# B&R Automation Studio project DuctLines (part 11)

#### Cyclic.ld
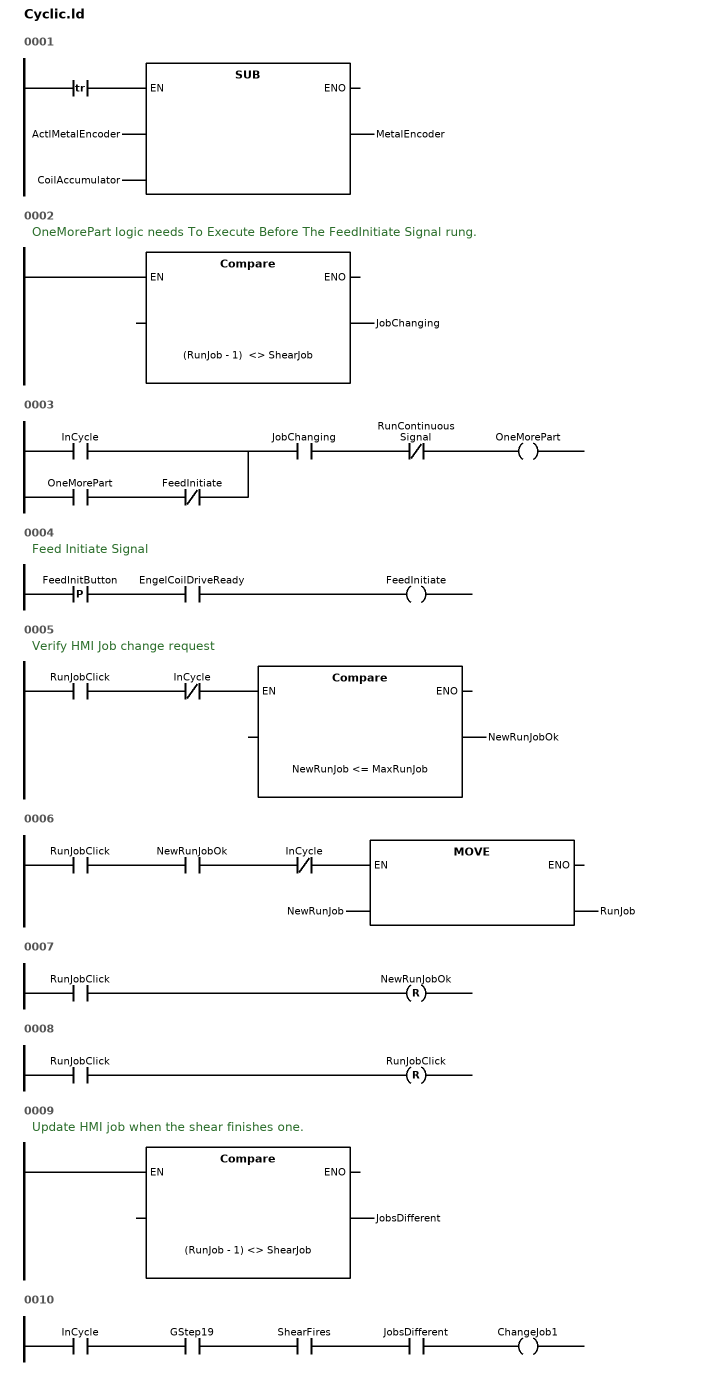
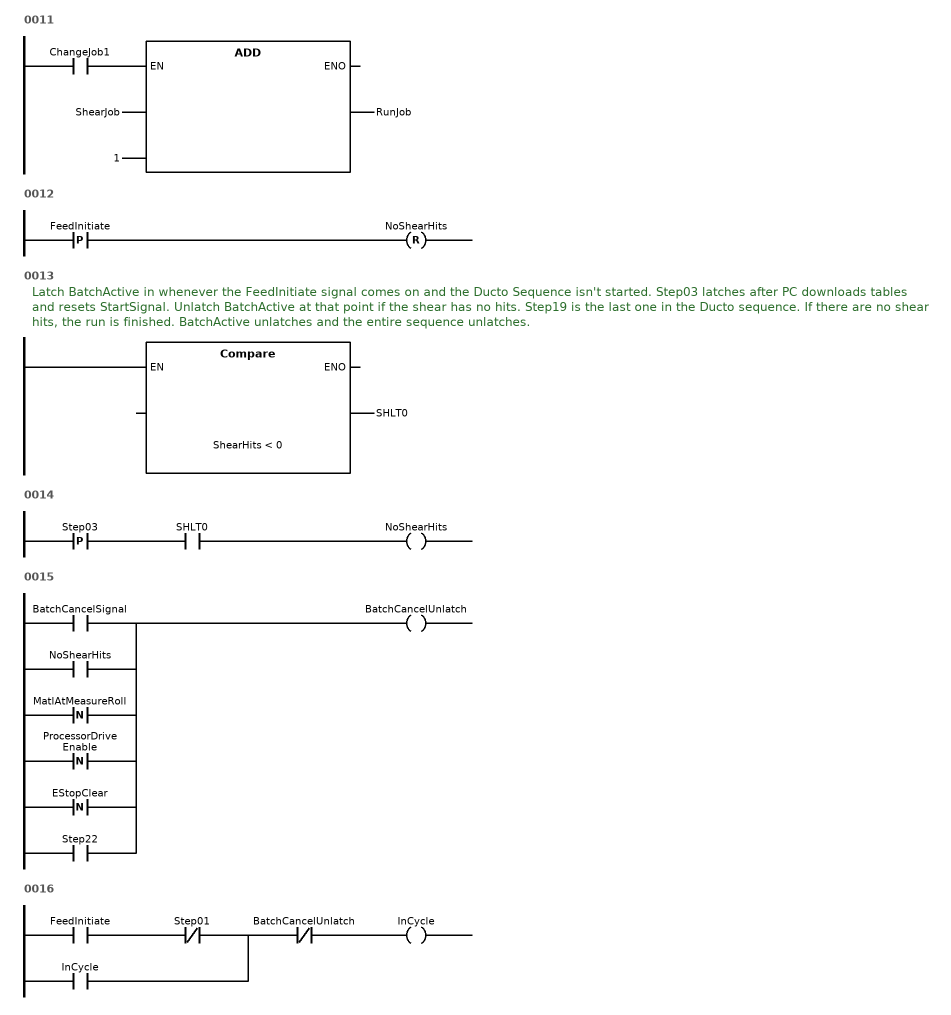
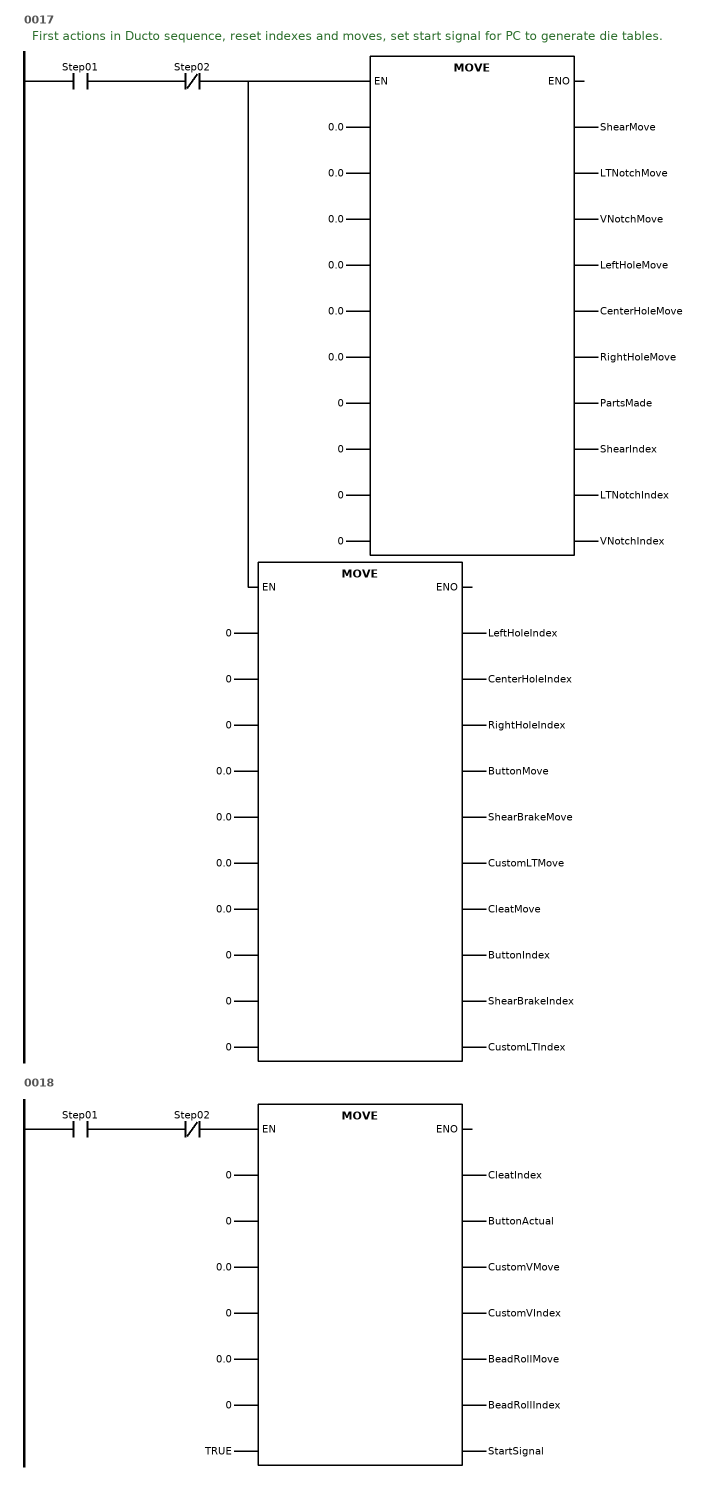
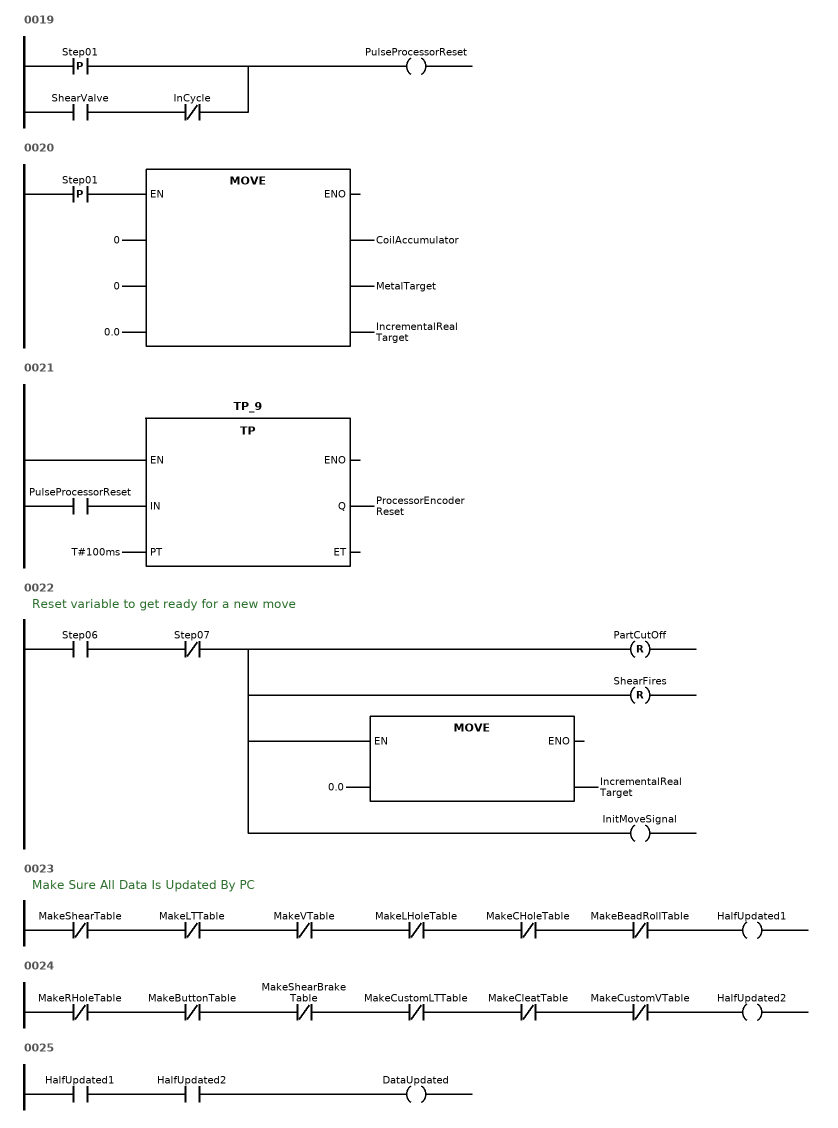
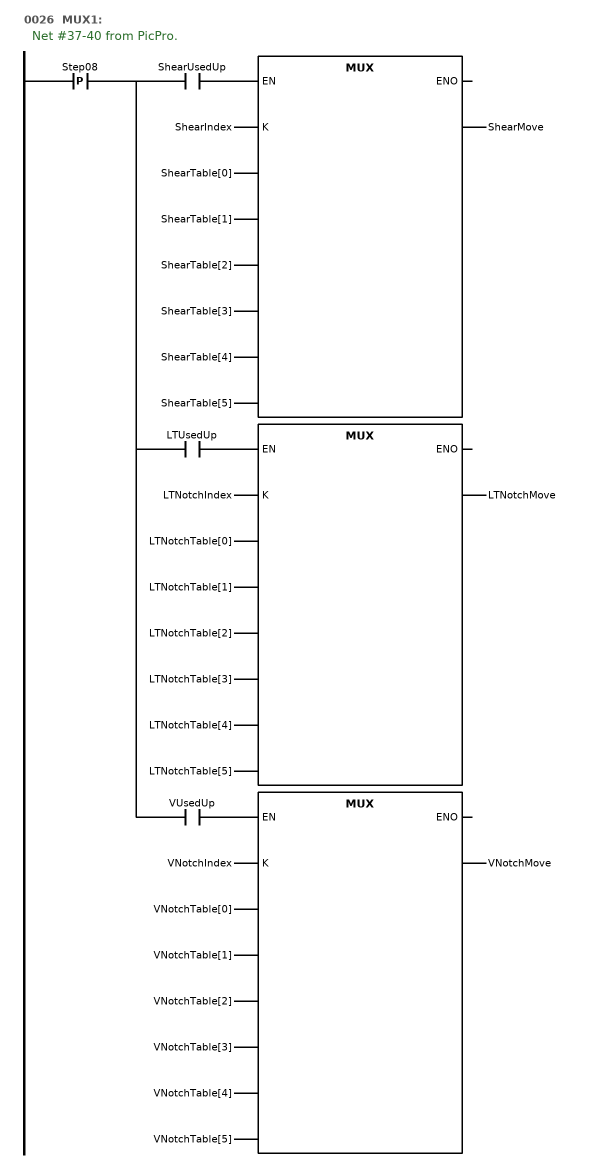
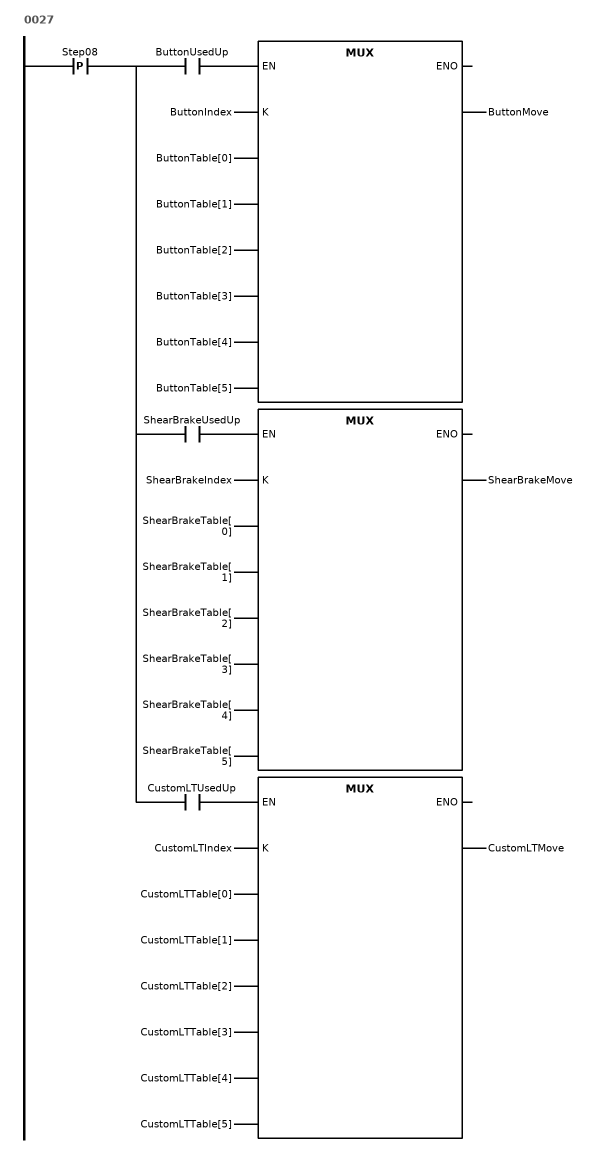
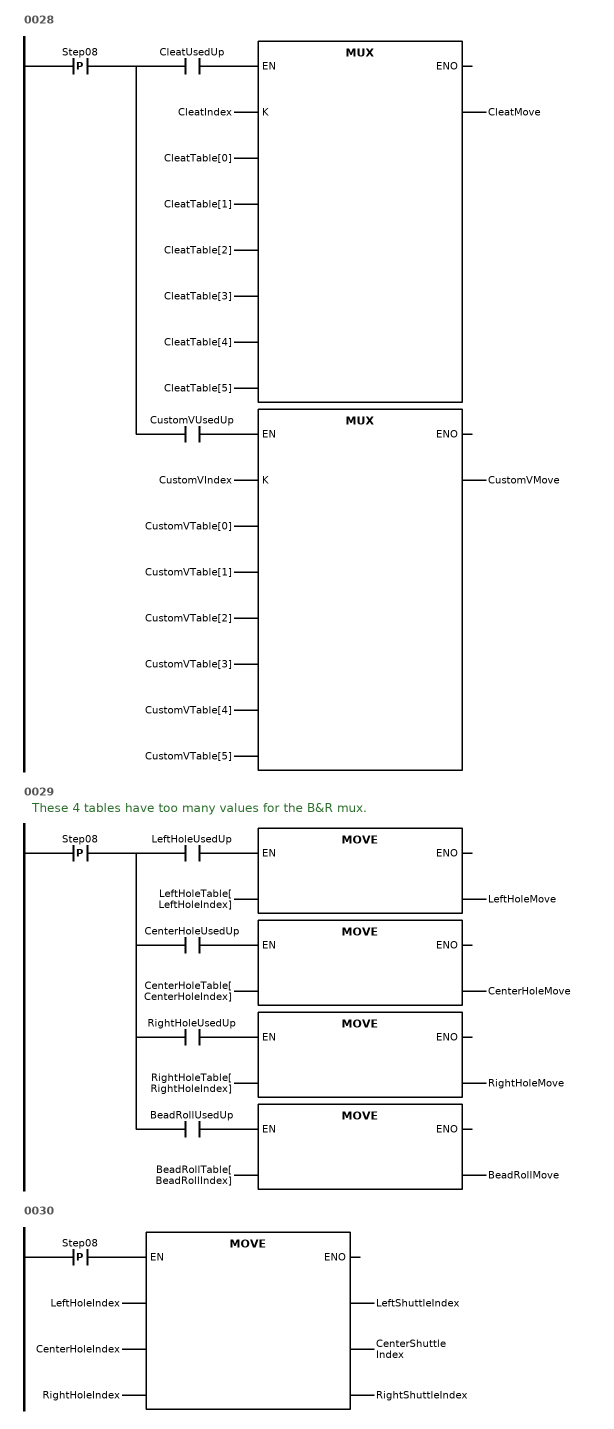
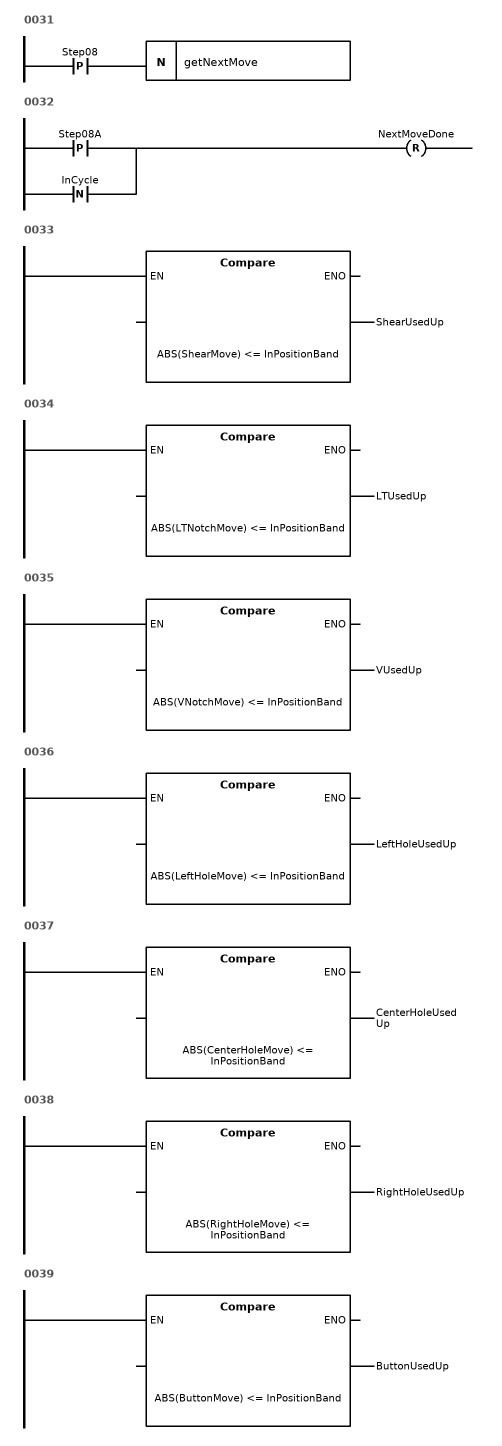
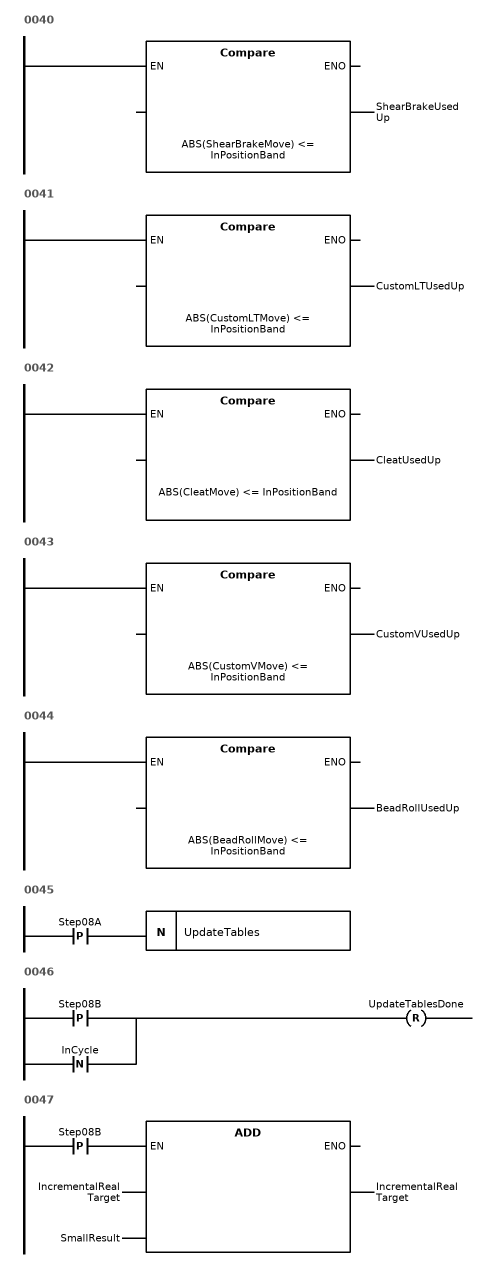
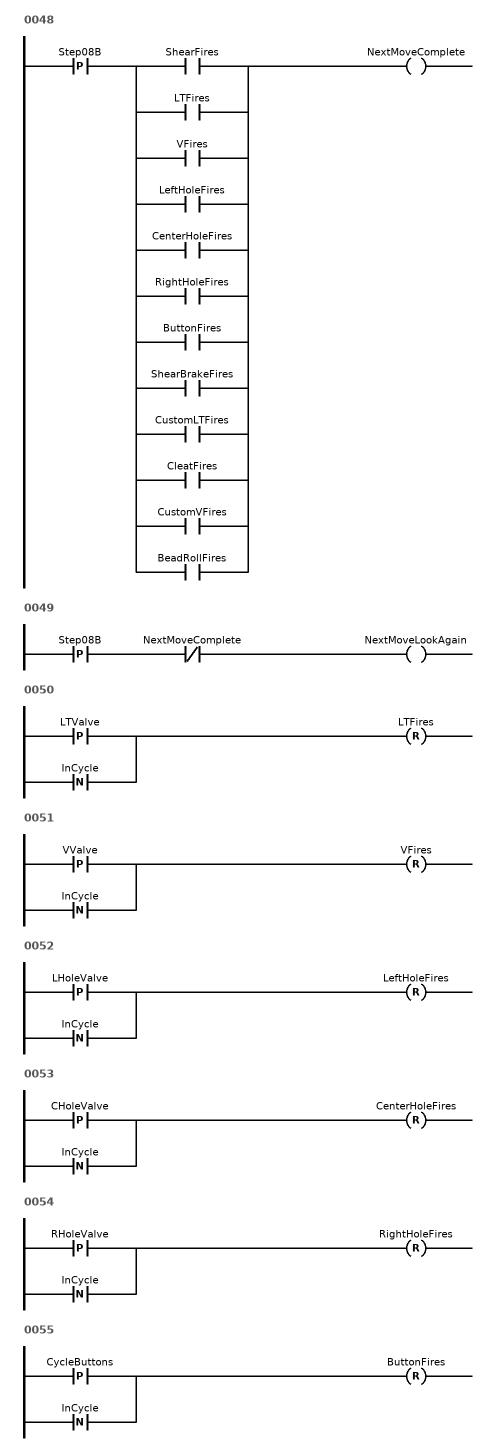
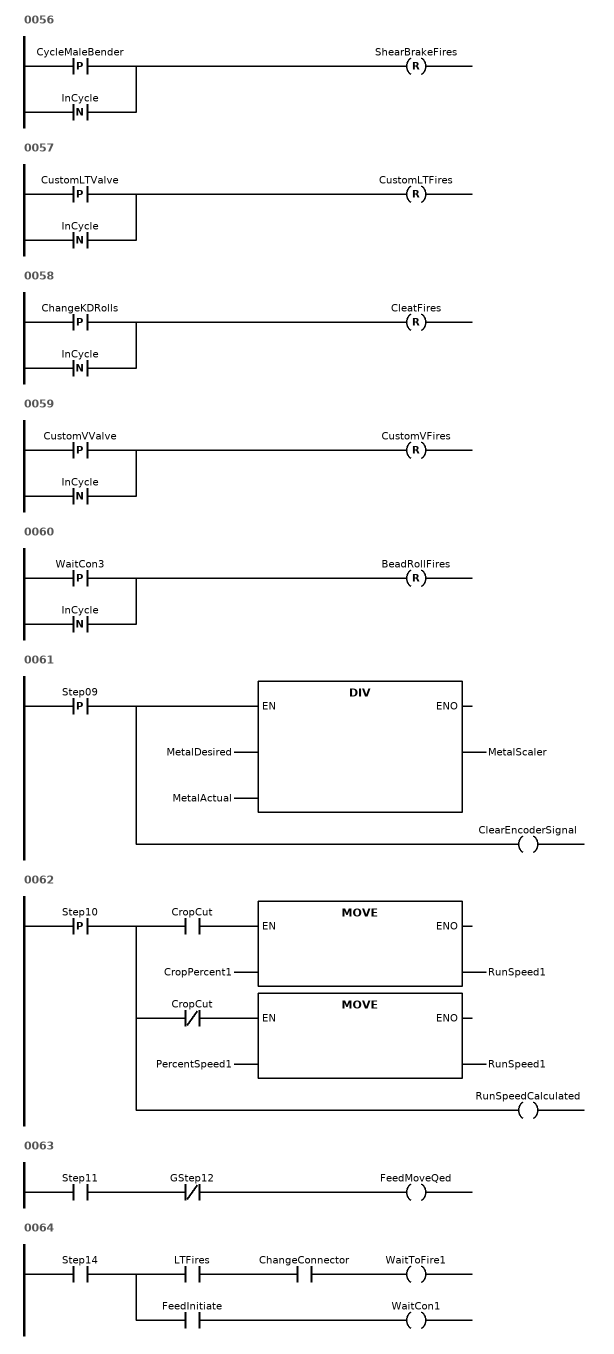
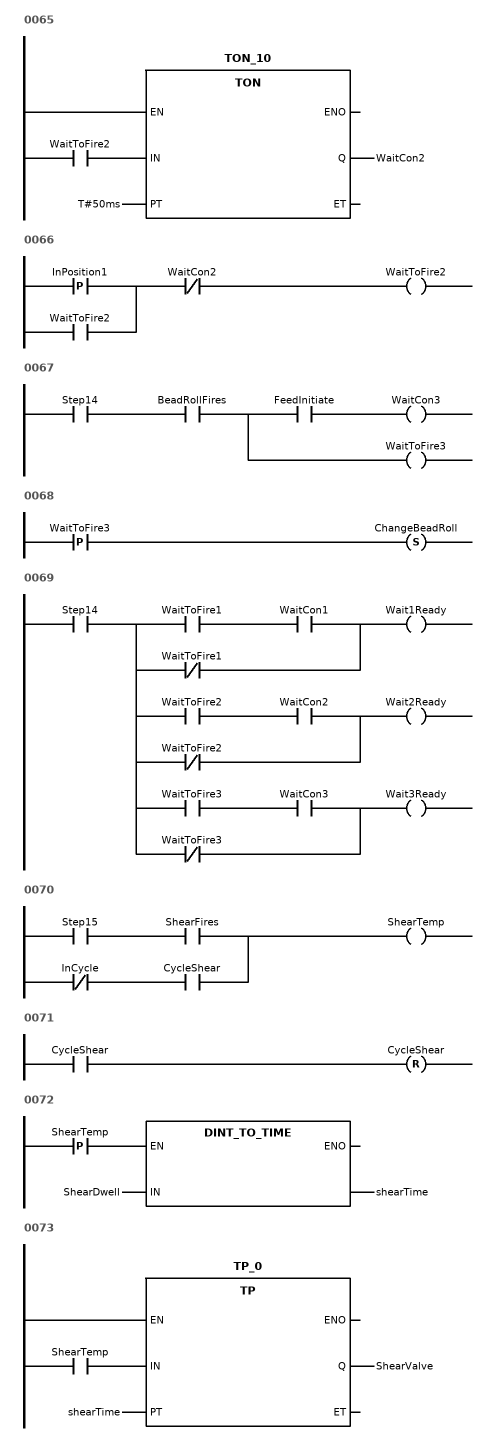
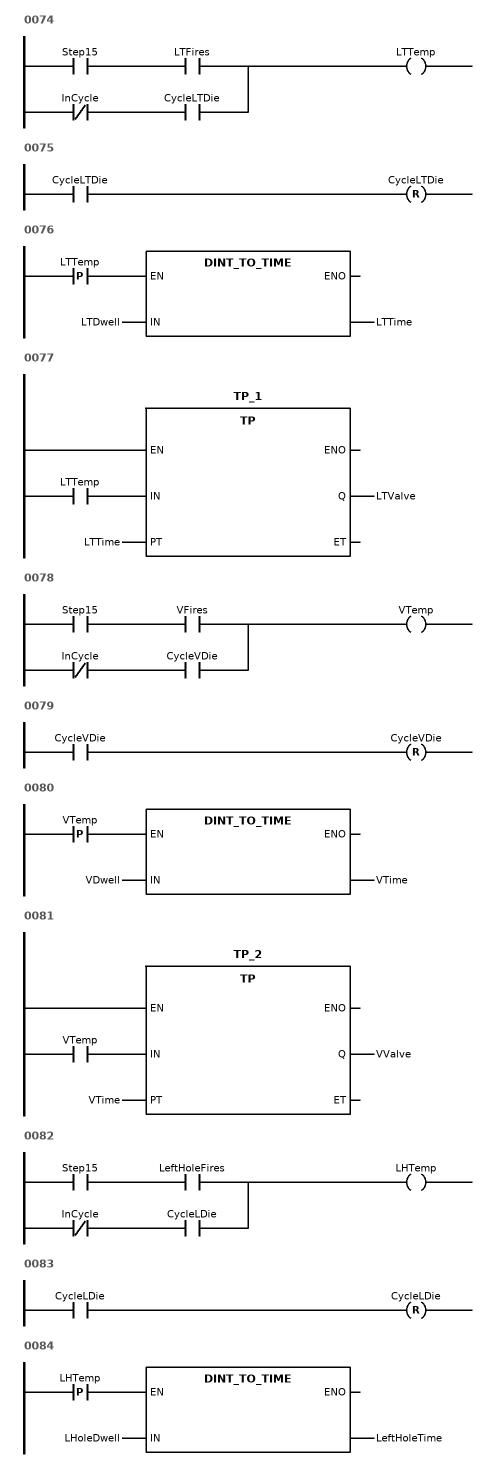
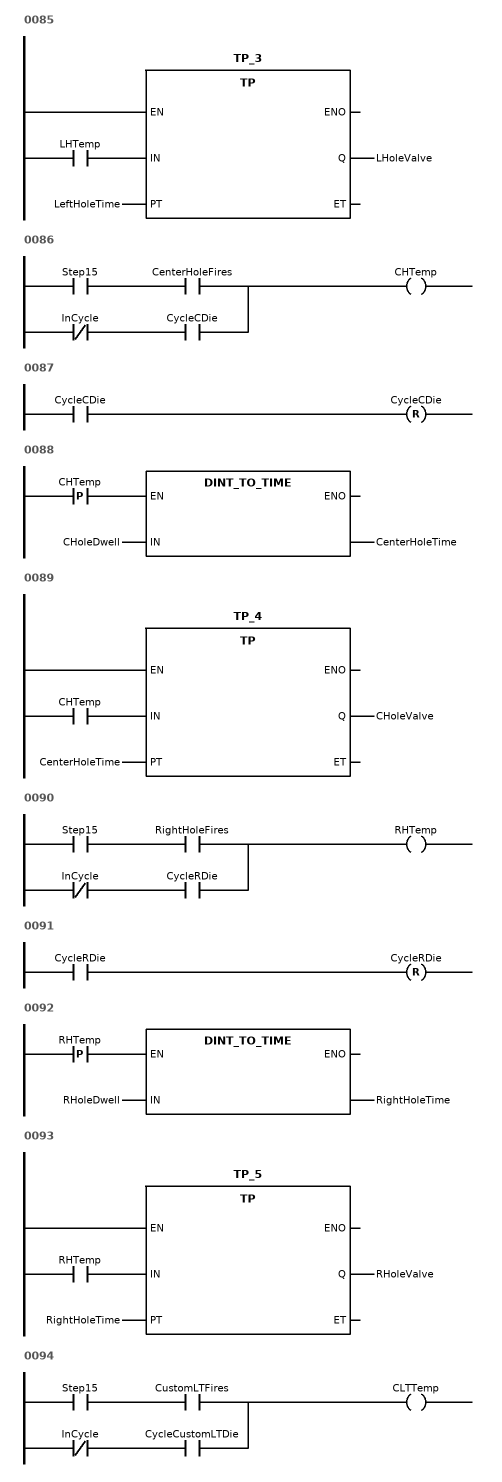
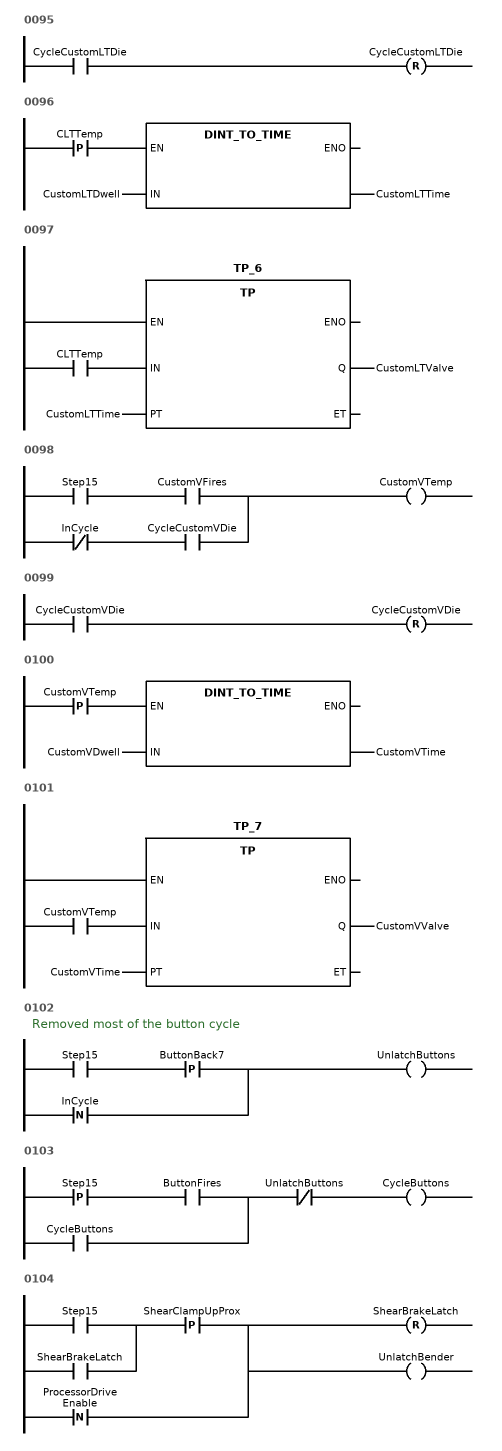
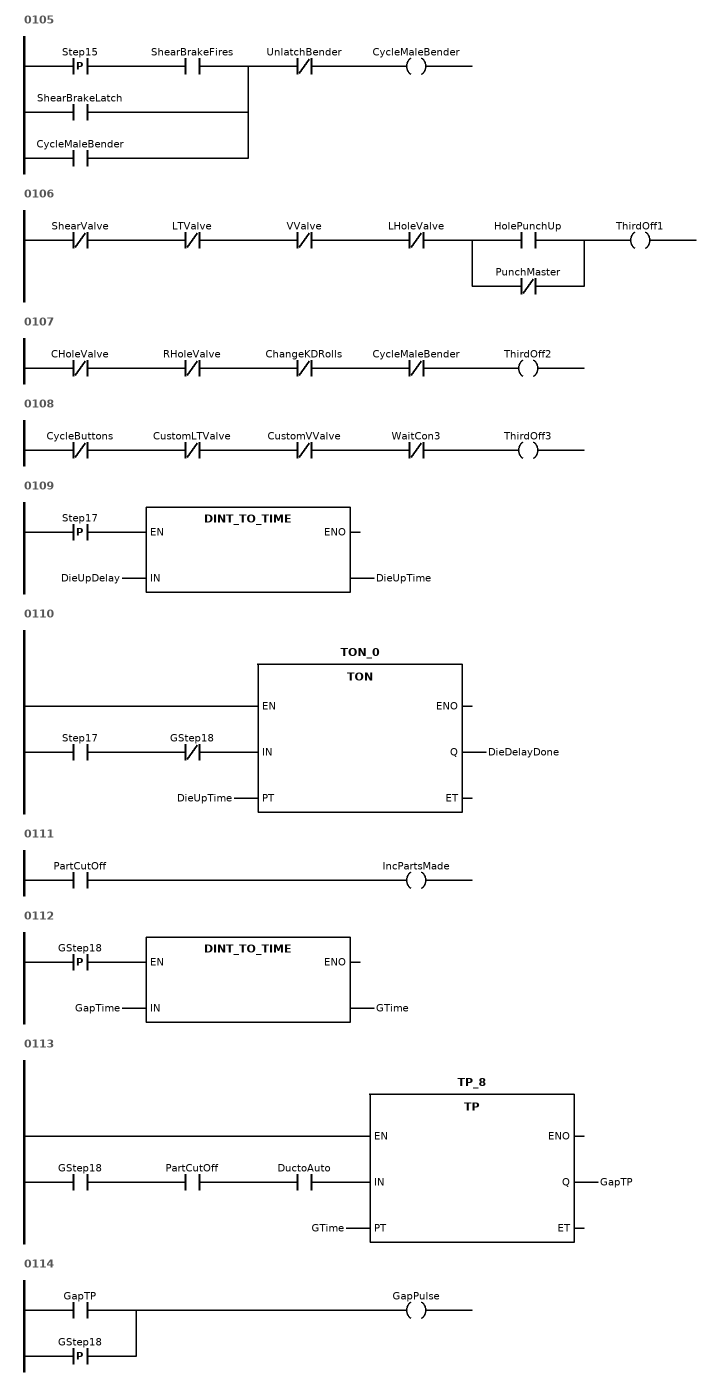
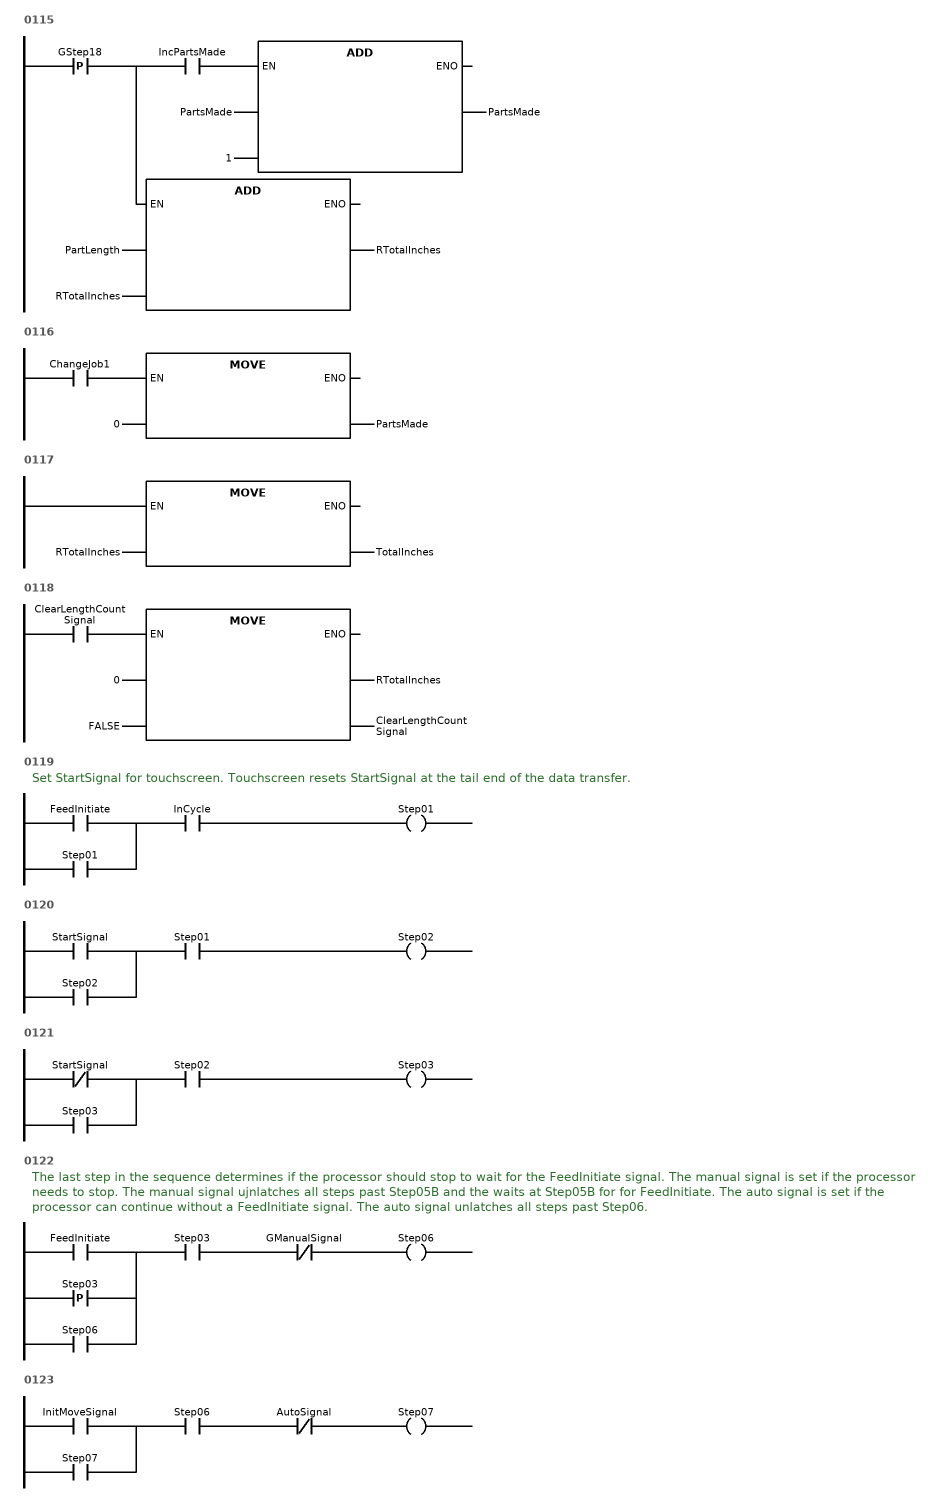
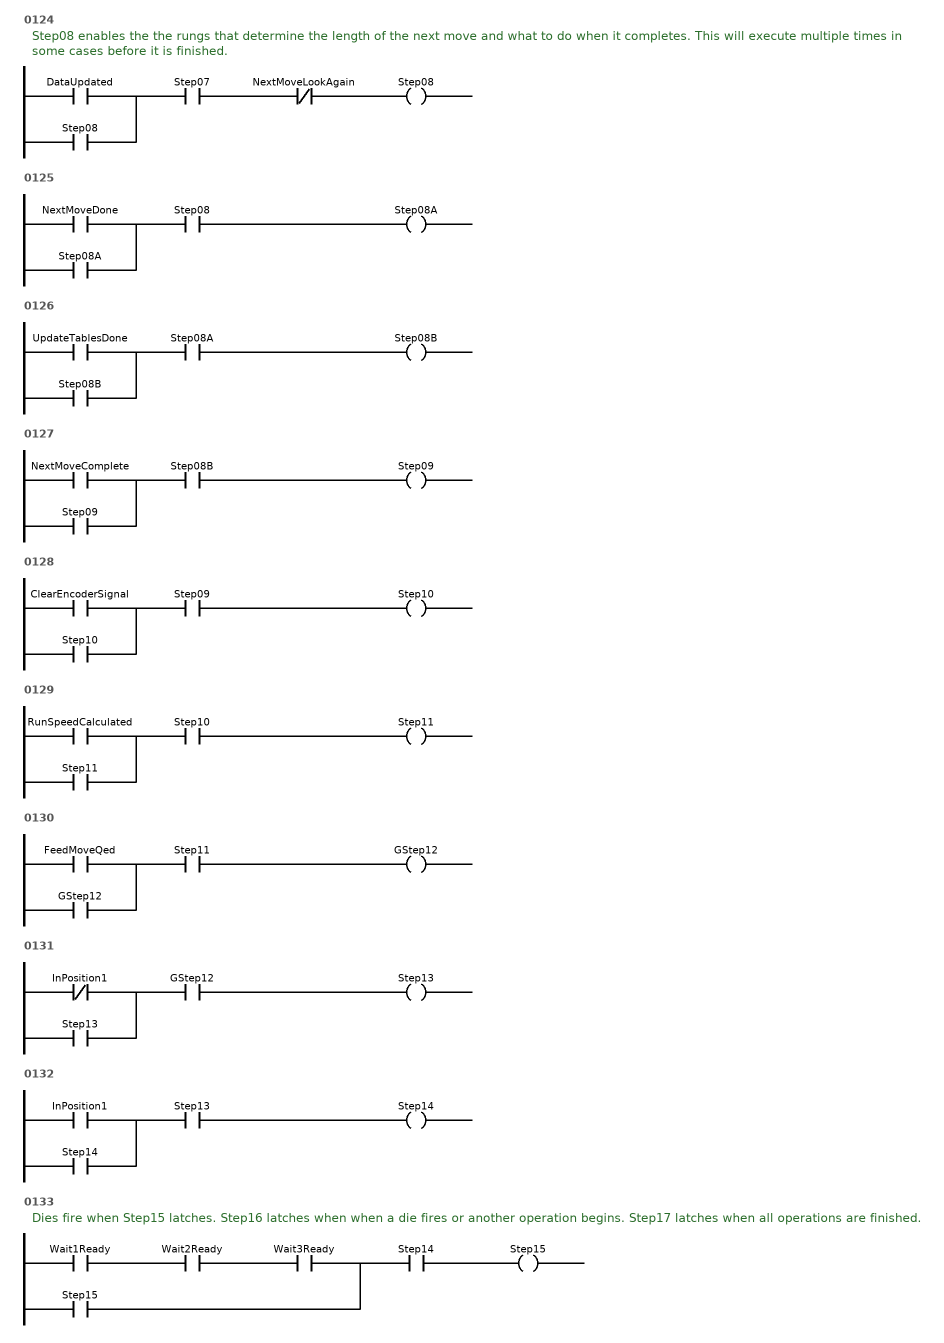
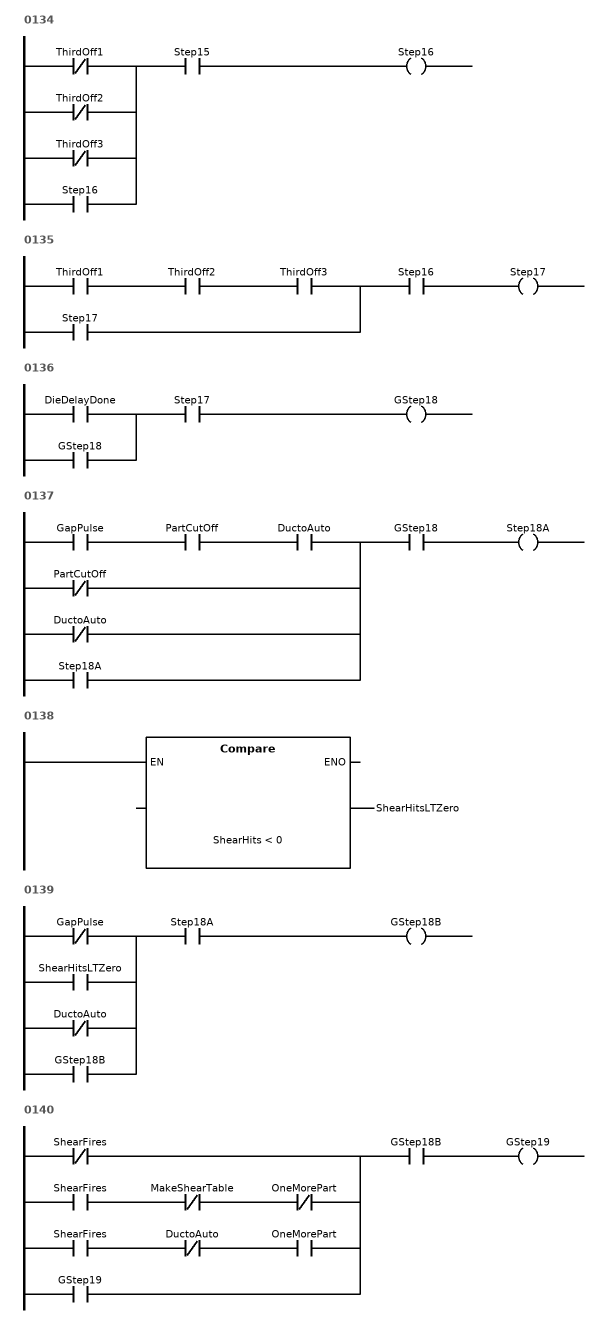
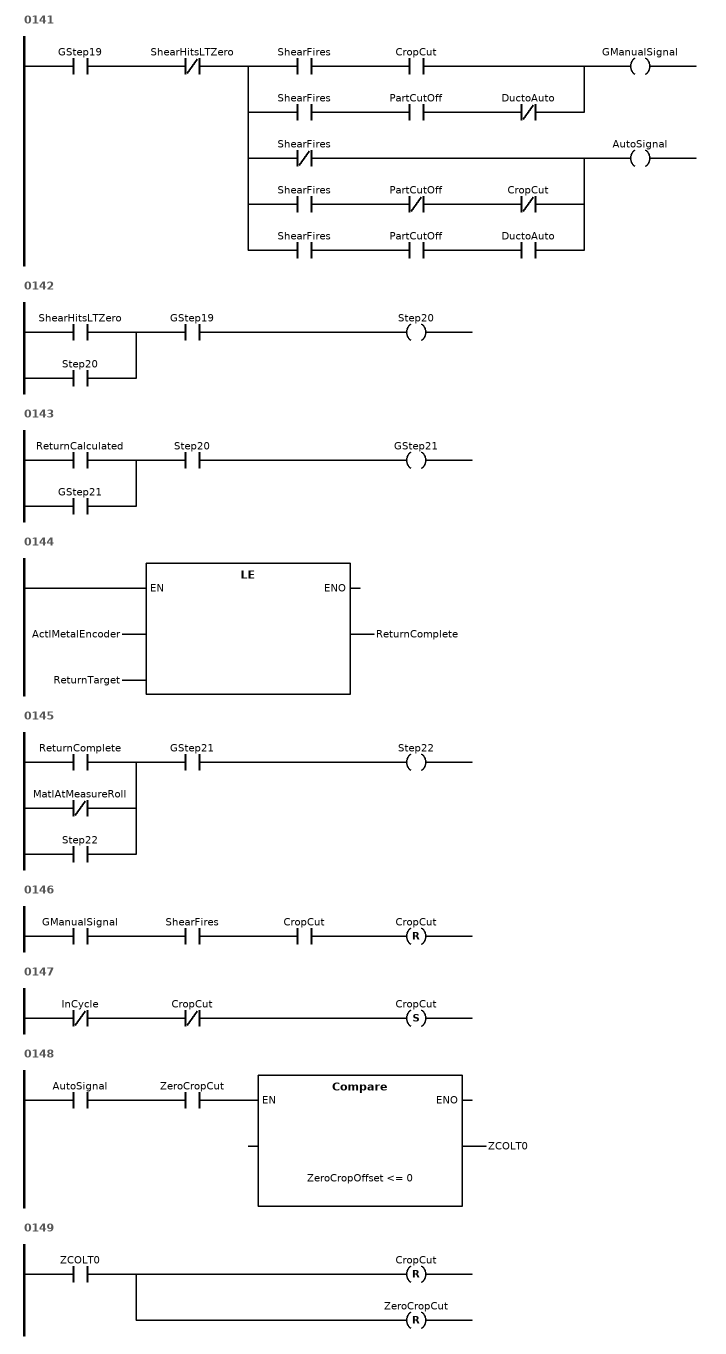
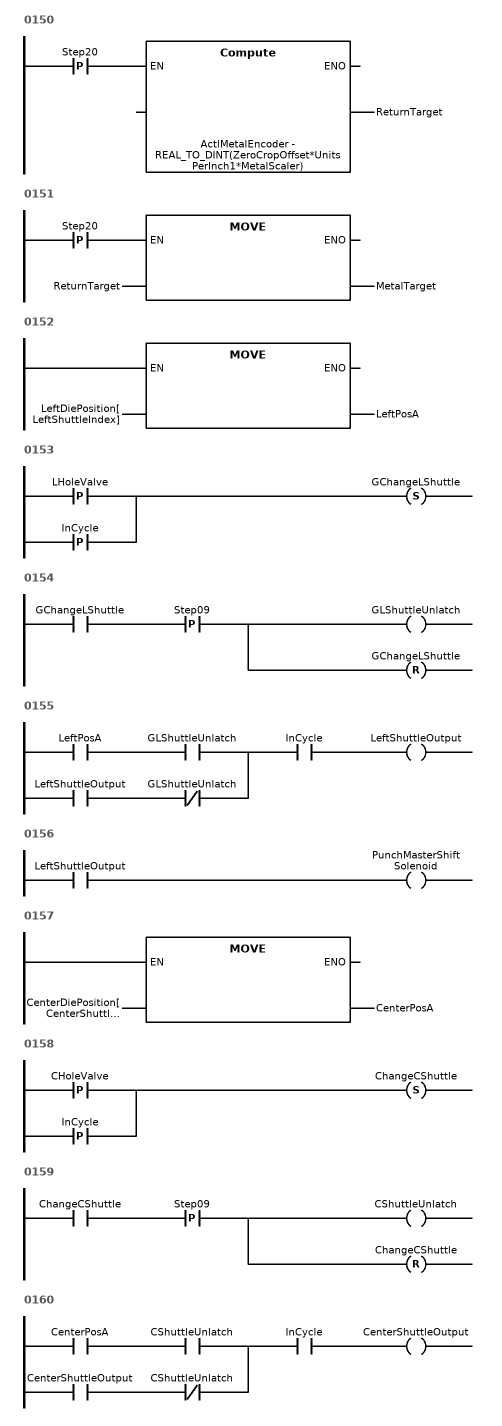
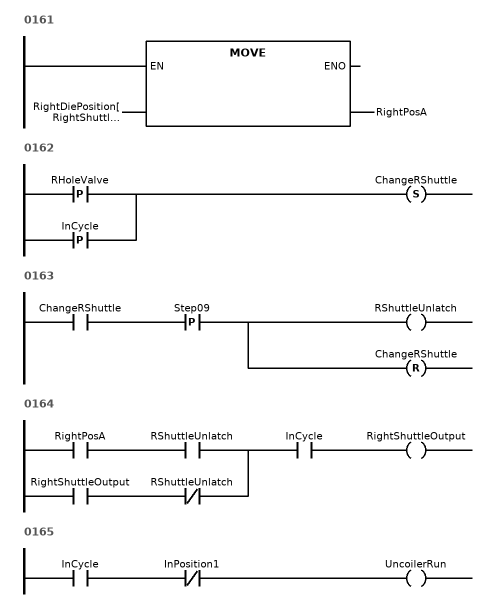
Ladder, written as Structured Text:
```iecst
PROGRAM _CYCLIC
VAR
    _e1 : R_TRIG;
    _e2 : R_TRIG;
    _e3 : R_TRIG;
    _e4 : F_TRIG;
    _e5 : F_TRIG;
    _e6 : F_TRIG;
    _e7 : R_TRIG;
    _e8 : R_TRIG;
    _e9 : R_TRIG;
    _e10 : R_TRIG;
    _e11 : R_TRIG;
    _e12 : R_TRIG;
    _e13 : R_TRIG;
    _e14 : R_TRIG;
    _e15 : R_TRIG;
    _e16 : F_TRIG;
    _e17 : R_TRIG;
    _e18 : R_TRIG;
    _e19 : F_TRIG;
    _e20 : R_TRIG;
    _e21 : R_TRIG;
    _e22 : R_TRIG;
    _e23 : R_TRIG;
    _e24 : F_TRIG;
    _e25 : R_TRIG;
    _e26 : F_TRIG;
    _e27 : R_TRIG;
    _e28 : F_TRIG;
    _e29 : R_TRIG;
    _e30 : F_TRIG;
    _e31 : R_TRIG;
    _e32 : F_TRIG;
    _e33 : R_TRIG;
    _e34 : F_TRIG;
    _e35 : R_TRIG;
    _e36 : F_TRIG;
    _e37 : R_TRIG;
    _e38 : F_TRIG;
    _e39 : R_TRIG;
    _e40 : F_TRIG;
    _e41 : R_TRIG;
    _e42 : F_TRIG;
    _e43 : R_TRIG;
    _e44 : F_TRIG;
    _e45 : R_TRIG;
    _e46 : R_TRIG;
    _e47 : R_TRIG;
    _e48 : R_TRIG;
    _e49 : R_TRIG;
    _e50 : R_TRIG;
    _e51 : R_TRIG;
    _e52 : R_TRIG;
    _e53 : R_TRIG;
    _e54 : R_TRIG;
    _e55 : R_TRIG;
    _e56 : R_TRIG;
    _e57 : R_TRIG;
    _e58 : F_TRIG;
    _e59 : R_TRIG;
    _e60 : R_TRIG;
    _e61 : F_TRIG;
    _p62 : BOOL;
    _e63 : R_TRIG;
    _p64 : BOOL;
    _e65 : R_TRIG;
    _e66 : R_TRIG;
    _e67 : R_TRIG;
    _e68 : R_TRIG;
    _p69 : BOOL;
    _e70 : R_TRIG;
    _e71 : R_TRIG;
    _e72 : R_TRIG;
    _e73 : R_TRIG;
    _e74 : R_TRIG;
    _e75 : R_TRIG;
    _e76 : R_TRIG;
    _e77 : R_TRIG;
    _e78 : R_TRIG;
    _e79 : R_TRIG;
    _e80 : R_TRIG;
    _e81 : R_TRIG;
END_VAR
(* Network 1 *)
MetalEncoder := ActlMetalEncoder - CoilAccumulator;

(* Network 2: OneMorePart logic needs To Execute Before The FeedInitiate Signal rung. *)
JobChanging := (RunJob - 1)  <> ShearJob;

(* Network 3 *)
OneMorePart := (InCycle OR (OneMorePart AND NOT FeedInitiate)) AND JobChanging AND NOT RunContinuousSignal;

(* Network 4: Feed Initiate Signal *)
_e1(CLK := FeedInitButton);
FeedInitiate := _e1.Q AND EngelCoilDriveReady;

(* Network 5: Verify HMI Job change request *)
IF RunJobClick AND NOT InCycle THEN NewRunJobOk := NewRunJob <= MaxRunJob; END_IF;

(* Network 6 *)
IF RunJobClick AND NewRunJobOk AND NOT InCycle THEN RunJob := NewRunJob; END_IF;

(* Network 7 *)
IF RunJobClick THEN NewRunJobOk := FALSE; END_IF;

(* Network 8 *)
IF RunJobClick THEN RunJobClick := FALSE; END_IF;

(* Network 9: Update HMI job when the shear finishes one. *)
JobsDifferent := (RunJob - 1) <> ShearJob;

(* Network 10 *)
ChangeJob1 := InCycle AND GStep19 AND ShearFires AND JobsDifferent;

(* Network 11 *)
IF ChangeJob1 THEN RunJob := ShearJob + 1; END_IF;

(* Network 12 *)
_e2(CLK := FeedInitiate);
IF _e2.Q THEN NoShearHits := FALSE; END_IF;

(* Network 13: Latch BatchActive in whenever the FeedInitiate signal comes on and the Ducto Sequence isn't started. Step03 latches after PC downloads tables and resets StartSignal. Unlatch BatchActive at that point if the shear has no hits. Step19 is the last one in the Ducto sequence. If there are no shear hits, the run is finished. BatchActive unlatches and the entire sequence unlatches. *)
SHLT0 := ShearHits < 0;

(* Network 14 *)
_e3(CLK := Step03);
NoShearHits := _e3.Q AND SHLT0;

(* Network 15 *)
_e4(CLK := MatlAtMeasureRoll);
_e5(CLK := ProcessorDriveEnable);
_e6(CLK := EStopClear);
BatchCancelUnlatch := BatchCancelSignal OR NoShearHits OR _e4.Q OR _e5.Q OR _e6.Q OR Step22;

(* Network 16 *)
InCycle := ((FeedInitiate AND NOT Step01) OR InCycle) AND NOT BatchCancelUnlatch;

(* Network 17: First actions in Ducto sequence, reset indexes and moves, set start signal for PC to generate die tables. *)
IF Step01 AND NOT Step02 THEN
    ShearMove := 0.0;
    LTNotchMove := 0.0;
    VNotchMove := 0.0;
    LeftHoleMove := 0.0;
    CenterHoleMove := 0.0;
    RightHoleMove := 0.0;
    PartsMade := 0;
    ShearIndex := 0;
    LTNotchIndex := 0;
    VNotchIndex := 0;
    LeftHoleIndex := 0;
    CenterHoleIndex := 0;
    RightHoleIndex := 0;
    ButtonMove := 0.0;
    ShearBrakeMove := 0.0;
    CustomLTMove := 0.0;
    CleatMove := 0.0;
    ButtonIndex := 0;
    ShearBrakeIndex := 0;
    CustomLTIndex := 0;
END_IF;

(* Network 18 *)
IF Step01 AND NOT Step02 THEN
    CleatIndex := 0;
    ButtonActual := 0;
    CustomVMove := 0.0;
    CustomVIndex := 0;
    BeadRollMove := 0.0;
    BeadRollIndex := 0;
    StartSignal := TRUE;
END_IF;

(* Network 19 *)
_e7(CLK := Step01);
PulseProcessorReset := _e7.Q OR (ShearValve AND NOT InCycle);

(* Network 20 *)
_e8(CLK := Step01);
IF _e8.Q THEN
    CoilAccumulator := 0;
    MetalTarget := 0;
    IncrementalRealTarget := 0.0;
END_IF;

(* Network 21 *)
TP_9(IN := PulseProcessorReset, PT := T#100ms);
ProcessorEncoderReset := TP_9.Q;

(* Network 22: Reset variable to get ready for a new move *)
IF Step06 AND NOT Step07 THEN
    PartCutOff := FALSE;
    ShearFires := FALSE;
    IncrementalRealTarget := 0.0;
END_IF;
InitMoveSignal := Step06 AND NOT Step07;

(* Network 23: Make Sure All Data Is Updated By PC *)
HalfUpdated1 := NOT MakeShearTable AND NOT MakeLTTable AND NOT MakeVTable AND NOT MakeLHoleTable AND NOT MakeCHoleTable AND NOT MakeBeadRollTable;

(* Network 24 *)
HalfUpdated2 := NOT MakeRHoleTable AND NOT MakeButtonTable AND NOT MakeShearBrakeTable AND NOT MakeCustomLTTable AND NOT MakeCleatTable AND NOT MakeCustomVTable;

(* Network 25 *)
DataUpdated := HalfUpdated1 AND HalfUpdated2;

(* Network 26: Net #37-40 from PicPro.  *)
MUX1:
_e9(CLK := Step08);
IF _e9.Q AND ShearUsedUp THEN
    ShearMove := MUX(K := ShearIndex, IN2 := ShearTable[0], IN3 := ShearTable[1], IN4 := ShearTable[2], IN5 := ShearTable[3], IN6 := ShearTable[4], IN7 := ShearTable[5]);
END_IF;
IF _e9.Q AND LTUsedUp THEN
    LTNotchMove := MUX(K := LTNotchIndex, IN2 := LTNotchTable[0], IN3 := LTNotchTable[1], IN4 := LTNotchTable[2], IN5 := LTNotchTable[3], IN6 := LTNotchTable[4], IN7 := LTNotchTable[5]);
END_IF;
IF _e9.Q AND VUsedUp THEN
    VNotchMove := MUX(K := VNotchIndex, IN2 := VNotchTable[0], IN3 := VNotchTable[1], IN4 := VNotchTable[2], IN5 := VNotchTable[3], IN6 := VNotchTable[4], IN7 := VNotchTable[5]);
END_IF;

(* Network 27 *)
_e10(CLK := Step08);
IF _e10.Q AND ButtonUsedUp THEN
    ButtonMove := MUX(K := ButtonIndex, IN2 := ButtonTable[0], IN3 := ButtonTable[1], IN4 := ButtonTable[2], IN5 := ButtonTable[3], IN6 := ButtonTable[4], IN7 := ButtonTable[5]);
END_IF;
IF _e10.Q AND ShearBrakeUsedUp THEN
    ShearBrakeMove := MUX(K := ShearBrakeIndex, IN2 := ShearBrakeTable[0], IN3 := ShearBrakeTable[1], IN4 := ShearBrakeTable[2], IN5 := ShearBrakeTable[3], IN6 := ShearBrakeTable[4], IN7 := ShearBrakeTable[5]);
END_IF;
IF _e10.Q AND CustomLTUsedUp THEN
    CustomLTMove := MUX(K := CustomLTIndex, IN2 := CustomLTTable[0], IN3 := CustomLTTable[1], IN4 := CustomLTTable[2], IN5 := CustomLTTable[3], IN6 := CustomLTTable[4], IN7 := CustomLTTable[5]);
END_IF;

(* Network 28 *)
_e11(CLK := Step08);
IF _e11.Q AND CleatUsedUp THEN
    CleatMove := MUX(K := CleatIndex, IN2 := CleatTable[0], IN3 := CleatTable[1], IN4 := CleatTable[2], IN5 := CleatTable[3], IN6 := CleatTable[4], IN7 := CleatTable[5]);
END_IF;
IF _e11.Q AND CustomVUsedUp THEN
    CustomVMove := MUX(K := CustomVIndex, IN2 := CustomVTable[0], IN3 := CustomVTable[1], IN4 := CustomVTable[2], IN5 := CustomVTable[3], IN6 := CustomVTable[4], IN7 := CustomVTable[5]);
END_IF;

(* Network 29: These 4 tables have too many values for the B&R mux. *)
_e12(CLK := Step08);
IF _e12.Q AND LeftHoleUsedUp THEN LeftHoleMove := LeftHoleTable[LeftHoleIndex]; END_IF;
IF _e12.Q AND CenterHoleUsedUp THEN CenterHoleMove := CenterHoleTable[CenterHoleIndex]; END_IF;
IF _e12.Q AND RightHoleUsedUp THEN RightHoleMove := RightHoleTable[RightHoleIndex]; END_IF;
IF _e12.Q AND BeadRollUsedUp THEN BeadRollMove := BeadRollTable[BeadRollIndex]; END_IF;

(* Network 30 *)
_e13(CLK := Step08);
IF _e13.Q THEN
    LeftShuttleIndex := LeftHoleIndex;
    CenterShuttleIndex := CenterHoleIndex;
    RightShuttleIndex := RightHoleIndex;
END_IF;

(* Network 31 *)
_e14(CLK := Step08);
IF _e14.Q THEN getNextMove; END_IF;

(* Network 32 *)
_e15(CLK := Step08A);
_e16(CLK := InCycle);
IF _e15.Q OR _e16.Q THEN NextMoveDone := FALSE; END_IF;

(* Network 33 *)
ShearUsedUp := ABS(ShearMove) <= InPositionBand;

(* Network 34 *)
LTUsedUp := ABS(LTNotchMove) <= InPositionBand;

(* Network 35 *)
VUsedUp := ABS(VNotchMove) <= InPositionBand;

(* Network 36 *)
LeftHoleUsedUp := ABS(LeftHoleMove) <= InPositionBand;

(* Network 37 *)
CenterHoleUsedUp := ABS(CenterHoleMove) <= InPositionBand;

(* Network 38 *)
RightHoleUsedUp := ABS(RightHoleMove) <= InPositionBand;

(* Network 39 *)
ButtonUsedUp := ABS(ButtonMove) <= InPositionBand;

(* Network 40 *)
ShearBrakeUsedUp := ABS(ShearBrakeMove) <= InPositionBand;

(* Network 41 *)
CustomLTUsedUp := ABS(CustomLTMove) <= InPositionBand;

(* Network 42 *)
CleatUsedUp := ABS(CleatMove) <= InPositionBand;

(* Network 43 *)
CustomVUsedUp := ABS(CustomVMove) <= InPositionBand;

(* Network 44 *)
BeadRollUsedUp := ABS(BeadRollMove) <= InPositionBand;

(* Network 45 *)
_e17(CLK := Step08A);
IF _e17.Q THEN UpdateTables; END_IF;

(* Network 46 *)
_e18(CLK := Step08B);
_e19(CLK := InCycle);
IF _e18.Q OR _e19.Q THEN UpdateTablesDone := FALSE; END_IF;

(* Network 47 *)
_e20(CLK := Step08B);
IF _e20.Q THEN IncrementalRealTarget := IncrementalRealTarget + SmallResult; END_IF;

(* Network 48 *)
_e21(CLK := Step08B);
NextMoveComplete := _e21.Q AND (ShearFires OR LTFires OR VFires OR LeftHoleFires OR CenterHoleFires OR RightHoleFires OR ButtonFires OR ShearBrakeFires OR CustomLTFires OR CleatFires OR CustomVFires OR BeadRollFires);

(* Network 49 *)
_e22(CLK := Step08B);
NextMoveLookAgain := _e22.Q AND NOT NextMoveComplete;

(* Network 50 *)
_e23(CLK := LTValve);
_e24(CLK := InCycle);
IF _e23.Q OR _e24.Q THEN LTFires := FALSE; END_IF;

(* Network 51 *)
_e25(CLK := VValve);
_e26(CLK := InCycle);
IF _e25.Q OR _e26.Q THEN VFires := FALSE; END_IF;

(* Network 52 *)
_e27(CLK := LHoleValve);
_e28(CLK := InCycle);
IF _e27.Q OR _e28.Q THEN LeftHoleFires := FALSE; END_IF;

(* Network 53 *)
_e29(CLK := CHoleValve);
_e30(CLK := InCycle);
IF _e29.Q OR _e30.Q THEN CenterHoleFires := FALSE; END_IF;

(* Network 54 *)
_e31(CLK := RHoleValve);
_e32(CLK := InCycle);
IF _e31.Q OR _e32.Q THEN RightHoleFires := FALSE; END_IF;

(* Network 55 *)
_e33(CLK := CycleButtons);
_e34(CLK := InCycle);
IF _e33.Q OR _e34.Q THEN ButtonFires := FALSE; END_IF;

(* Network 56 *)
_e35(CLK := CycleMaleBender);
_e36(CLK := InCycle);
IF _e35.Q OR _e36.Q THEN ShearBrakeFires := FALSE; END_IF;

(* Network 57 *)
_e37(CLK := CustomLTValve);
_e38(CLK := InCycle);
IF _e37.Q OR _e38.Q THEN CustomLTFires := FALSE; END_IF;

(* Network 58 *)
_e39(CLK := ChangeKDRolls);
_e40(CLK := InCycle);
IF _e39.Q OR _e40.Q THEN CleatFires := FALSE; END_IF;

(* Network 59 *)
_e41(CLK := CustomVValve);
_e42(CLK := InCycle);
IF _e41.Q OR _e42.Q THEN CustomVFires := FALSE; END_IF;

(* Network 60 *)
_e43(CLK := WaitCon3);
_e44(CLK := InCycle);
IF _e43.Q OR _e44.Q THEN BeadRollFires := FALSE; END_IF;

(* Network 61 *)
_e45(CLK := Step09);
IF _e45.Q THEN MetalScaler := MetalDesired / MetalActual; END_IF;
ClearEncoderSignal := _e45.Q;

(* Network 62 *)
_e46(CLK := Step10);
IF _e46.Q AND CropCut THEN RunSpeed1 := CropPercent1; END_IF;
IF _e46.Q AND NOT CropCut THEN RunSpeed1 := PercentSpeed1; END_IF;
RunSpeedCalculated := _e46.Q;

(* Network 63 *)
FeedMoveQed := Step11 AND NOT GStep12;

(* Network 64 *)
WaitToFire1 := Step14 AND LTFires AND ChangeConnector;
WaitCon1 := Step14 AND FeedInitiate;

(* Network 65 *)
TON_10(IN := WaitToFire2, PT := T#50ms);
WaitCon2 := TON_10.Q;

(* Network 66 *)
_e47(CLK := InPosition1);
WaitToFire2 := (_e47.Q OR WaitToFire2) AND NOT WaitCon2;

(* Network 67 *)
WaitCon3 := Step14 AND BeadRollFires AND FeedInitiate;
WaitToFire3 := Step14 AND BeadRollFires;

(* Network 68 *)
_e48(CLK := WaitToFire3);
IF _e48.Q THEN ChangeBeadRoll := TRUE; END_IF;

(* Network 69 *)
Wait1Ready := Step14 AND ((WaitToFire1 AND WaitCon1) OR NOT WaitToFire1);
Wait2Ready := Step14 AND ((WaitToFire2 AND WaitCon2) OR NOT WaitToFire2);
Wait3Ready := Step14 AND ((WaitToFire3 AND WaitCon3) OR NOT WaitToFire3);

(* Network 70 *)
ShearTemp := (Step15 AND ShearFires) OR (NOT InCycle AND CycleShear);

(* Network 71 *)
IF CycleShear THEN CycleShear := FALSE; END_IF;

(* Network 72 *)
_e49(CLK := ShearTemp);
IF _e49.Q THEN shearTime := DINT_TO_TIME(ShearDwell); END_IF;

(* Network 73 *)
TP_0(IN := ShearTemp, PT := shearTime);
ShearValve := TP_0.Q;

(* Network 74 *)
LTTemp := (Step15 AND LTFires) OR (NOT InCycle AND CycleLTDie);

(* Network 75 *)
IF CycleLTDie THEN CycleLTDie := FALSE; END_IF;

(* Network 76 *)
_e50(CLK := LTTemp);
IF _e50.Q THEN LTTime := DINT_TO_TIME(LTDwell); END_IF;

(* Network 77 *)
TP_1(IN := LTTemp, PT := LTTime);
LTValve := TP_1.Q;

(* Network 78 *)
VTemp := (Step15 AND VFires) OR (NOT InCycle AND CycleVDie);

(* Network 79 *)
IF CycleVDie THEN CycleVDie := FALSE; END_IF;

(* Network 80 *)
_e51(CLK := VTemp);
IF _e51.Q THEN VTime := DINT_TO_TIME(VDwell); END_IF;

(* Network 81 *)
TP_2(IN := VTemp, PT := VTime);
VValve := TP_2.Q;

(* Network 82 *)
LHTemp := (Step15 AND LeftHoleFires) OR (NOT InCycle AND CycleLDie);

(* Network 83 *)
IF CycleLDie THEN CycleLDie := FALSE; END_IF;

(* Network 84 *)
_e52(CLK := LHTemp);
IF _e52.Q THEN LeftHoleTime := DINT_TO_TIME(LHoleDwell); END_IF;

(* Network 85 *)
TP_3(IN := LHTemp, PT := LeftHoleTime);
LHoleValve := TP_3.Q;

(* Network 86 *)
CHTemp := (Step15 AND CenterHoleFires) OR (NOT InCycle AND CycleCDie);

(* Network 87 *)
IF CycleCDie THEN CycleCDie := FALSE; END_IF;

(* Network 88 *)
_e53(CLK := CHTemp);
IF _e53.Q THEN CenterHoleTime := DINT_TO_TIME(CHoleDwell); END_IF;

(* Network 89 *)
TP_4(IN := CHTemp, PT := CenterHoleTime);
CHoleValve := TP_4.Q;

(* Network 90 *)
RHTemp := (Step15 AND RightHoleFires) OR (NOT InCycle AND CycleRDie);

(* Network 91 *)
IF CycleRDie THEN CycleRDie := FALSE; END_IF;

(* Network 92 *)
_e54(CLK := RHTemp);
IF _e54.Q THEN RightHoleTime := DINT_TO_TIME(RHoleDwell); END_IF;

(* Network 93 *)
TP_5(IN := RHTemp, PT := RightHoleTime);
RHoleValve := TP_5.Q;

(* Network 94 *)
CLTTemp := (Step15 AND CustomLTFires) OR (NOT InCycle AND CycleCustomLTDie);

(* Network 95 *)
IF CycleCustomLTDie THEN CycleCustomLTDie := FALSE; END_IF;

(* Network 96 *)
_e55(CLK := CLTTemp);
IF _e55.Q THEN CustomLTTime := DINT_TO_TIME(CustomLTDwell); END_IF;

(* Network 97 *)
TP_6(IN := CLTTemp, PT := CustomLTTime);
CustomLTValve := TP_6.Q;

(* Network 98 *)
CustomVTemp := (Step15 AND CustomVFires) OR (NOT InCycle AND CycleCustomVDie);

(* Network 99 *)
IF CycleCustomVDie THEN CycleCustomVDie := FALSE; END_IF;

(* Network 100 *)
_e56(CLK := CustomVTemp);
IF _e56.Q THEN CustomVTime := DINT_TO_TIME(CustomVDwell); END_IF;

(* Network 101 *)
TP_7(IN := CustomVTemp, PT := CustomVTime);
CustomVValve := TP_7.Q;

(* Network 102: Removed most of the button cycle *)
_e57(CLK := ButtonBack7);
_e58(CLK := InCycle);
UnlatchButtons := (Step15 AND _e57.Q) OR _e58.Q;

(* Network 103 *)
_e59(CLK := Step15);
CycleButtons := ((_e59.Q AND ButtonFires) OR CycleButtons) AND NOT UnlatchButtons;

(* Network 104 *)
_e60(CLK := ShearClampUpProx);
_e61(CLK := ProcessorDriveEnable);
_p62 := (Step15 OR ShearBrakeLatch) AND _e60.Q;
IF ((Step15 OR ShearBrakeLatch) AND _e60.Q) OR _e61.Q THEN ShearBrakeLatch := FALSE; END_IF;
UnlatchBender := _p62 OR _e61.Q;

(* Network 105 *)
_e63(CLK := Step15);
CycleMaleBender := ((_e63.Q AND ShearBrakeFires) OR ShearBrakeLatch OR CycleMaleBender) AND NOT UnlatchBender;

(* Network 106 *)
_p64 := NOT ShearValve AND NOT LTValve AND NOT VValve AND NOT LHoleValve;
ThirdOff1 := _p64 AND (HolePunchUp OR NOT PunchMaster);

(* Network 107 *)
ThirdOff2 := NOT CHoleValve AND NOT RHoleValve AND NOT ChangeKDRolls AND NOT CycleMaleBender;

(* Network 108 *)
ThirdOff3 := NOT CycleButtons AND NOT CustomLTValve AND NOT CustomVValve AND NOT WaitCon3;

(* Network 109 *)
_e65(CLK := Step17);
IF _e65.Q THEN DieUpTime := DINT_TO_TIME(DieUpDelay); END_IF;

(* Network 110 *)
TON_0(IN := Step17 AND NOT GStep18, PT := DieUpTime);
DieDelayDone := TON_0.Q;

(* Network 111 *)
IncPartsMade := PartCutOff;

(* Network 112 *)
_e66(CLK := GStep18);
IF _e66.Q THEN GTime := DINT_TO_TIME(GapTime); END_IF;

(* Network 113 *)
TP_8(IN := GStep18 AND PartCutOff AND DuctoAuto, PT := GTime);
GapTP := TP_8.Q;

(* Network 114 *)
_e67(CLK := GStep18);
GapPulse := GapTP OR _e67.Q;

(* Network 115 *)
_e68(CLK := GStep18);
IF _e68.Q AND IncPartsMade THEN PartsMade := PartsMade + 1; END_IF;
IF _e68.Q THEN RTotalInches := PartLength + RTotalInches; END_IF;

(* Network 116 *)
IF ChangeJob1 THEN PartsMade := 0; END_IF;

(* Network 117 *)
TotalInches := RTotalInches;

(* Network 118 *)
IF ClearLengthCountSignal THEN RTotalInches := 0; END_IF;
_p69 := ClearLengthCountSignal;
IF _p69 THEN ClearLengthCountSignal := FALSE; END_IF;

(* Network 119: Set StartSignal for touchscreen. Touchscreen resets StartSignal at the tail end of the data transfer. *)
Step01 := (FeedInitiate OR Step01) AND InCycle;

(* Network 120 *)
Step02 := (StartSignal OR Step02) AND Step01;

(* Network 121 *)
Step03 := (NOT StartSignal OR Step03) AND Step02;

(* Network 122: The last step in the sequence determines if the processor should stop to wait for the FeedInitiate signal. The manual signal is set if the processor needs to stop. The manual signal ujnlatches all steps past Step05B and the waits at Step05B for for FeedInitiate. The auto signal is set if the processor can continue without a FeedInitiate signal. The auto signal unlatches all steps past Step06. *)
_e70(CLK := Step03);
Step06 := (FeedInitiate OR _e70.Q OR Step06) AND Step03 AND NOT GManualSignal;

(* Network 123 *)
Step07 := (InitMoveSignal OR Step07) AND Step06 AND NOT AutoSignal;

(* Network 124: Step08 enables the the rungs that determine the length of the next move and what to do when it completes. This will execute multiple times in some cases before it is finished. *)
Step08 := (DataUpdated OR Step08) AND Step07 AND NOT NextMoveLookAgain;

(* Network 125 *)
Step08A := (NextMoveDone OR Step08A) AND Step08;

(* Network 126 *)
Step08B := (UpdateTablesDone OR Step08B) AND Step08A;

(* Network 127 *)
Step09 := (NextMoveComplete OR Step09) AND Step08B;

(* Network 128 *)
Step10 := (ClearEncoderSignal OR Step10) AND Step09;

(* Network 129 *)
Step11 := (RunSpeedCalculated OR Step11) AND Step10;

(* Network 130 *)
GStep12 := (FeedMoveQed OR GStep12) AND Step11;

(* Network 131 *)
Step13 := (NOT InPosition1 OR Step13) AND GStep12;

(* Network 132 *)
Step14 := (InPosition1 OR Step14) AND Step13;

(* Network 133: Dies fire when Step15 latches. Step16 latches when when a die fires or another operation begins. Step17 latches when all operations are finished. *)
Step15 := ((Wait1Ready AND Wait2Ready AND Wait3Ready) OR Step15) AND Step14;

(* Network 134 *)
Step16 := (NOT ThirdOff1 OR NOT ThirdOff2 OR NOT ThirdOff3 OR Step16) AND Step15;

(* Network 135 *)
Step17 := ((ThirdOff1 AND ThirdOff2 AND ThirdOff3) OR Step17) AND Step16;

(* Network 136 *)
GStep18 := (DieDelayDone OR GStep18) AND Step17;

(* Network 137 *)
Step18A := ((GapPulse AND PartCutOff AND DuctoAuto) OR NOT PartCutOff OR NOT DuctoAuto OR Step18A) AND GStep18;

(* Network 138 *)
ShearHitsLTZero := ShearHits < 0;

(* Network 139 *)
GStep18B := (NOT GapPulse OR ShearHitsLTZero OR NOT DuctoAuto OR GStep18B) AND Step18A;

(* Network 140 *)
GStep19 := (NOT ShearFires OR (ShearFires AND ((NOT MakeShearTable AND NOT OneMorePart) OR (NOT DuctoAuto AND OneMorePart))) OR GStep19) AND GStep18B;

(* Network 141 *)
GManualSignal := GStep19 AND NOT ShearHitsLTZero AND ShearFires AND (CropCut OR (PartCutOff AND NOT DuctoAuto));
AutoSignal := GStep19 AND NOT ShearHitsLTZero AND (NOT ShearFires OR (ShearFires AND ((NOT PartCutOff AND NOT CropCut) OR (PartCutOff AND DuctoAuto))));

(* Network 142 *)
Step20 := (ShearHitsLTZero OR Step20) AND GStep19;

(* Network 143 *)
GStep21 := (ReturnCalculated OR GStep21) AND Step20;

(* Network 144 *)
ReturnComplete := ActlMetalEncoder <= ReturnTarget;

(* Network 145 *)
Step22 := (ReturnComplete OR NOT MatlAtMeasureRoll OR Step22) AND GStep21;

(* Network 146 *)
IF GManualSignal AND ShearFires AND CropCut THEN CropCut := FALSE; END_IF;

(* Network 147 *)
IF NOT InCycle AND NOT CropCut THEN CropCut := TRUE; END_IF;

(* Network 148 *)
IF AutoSignal AND ZeroCropCut THEN ZCOLT0 := ZeroCropOffset <= 0; END_IF;

(* Network 149 *)
IF ZCOLT0 THEN
    CropCut := FALSE;
    ZeroCropCut := FALSE;
END_IF;

(* Network 150 *)
_e71(CLK := Step20);
IF _e71.Q THEN
    ReturnTarget := ActlMetalEncoder - REAL_TO_DINT(ZeroCropOffset*UnitsPerInch1*MetalScaler);
END_IF;

(* Network 151 *)
_e72(CLK := Step20);
IF _e72.Q THEN MetalTarget := ReturnTarget; END_IF;

(* Network 152 *)
LeftPosA := LeftDiePosition[LeftShuttleIndex];

(* Network 153 *)
_e73(CLK := LHoleValve);
_e74(CLK := InCycle);
IF _e73.Q OR _e74.Q THEN GChangeLShuttle := TRUE; END_IF;

(* Network 154 *)
_e75(CLK := Step09);
GLShuttleUnlatch := GChangeLShuttle AND _e75.Q;
IF GChangeLShuttle AND _e75.Q THEN GChangeLShuttle := FALSE; END_IF;

(* Network 155 *)
LeftShuttleOutput := ((LeftPosA AND GLShuttleUnlatch) OR (LeftShuttleOutput AND NOT GLShuttleUnlatch)) AND InCycle;

(* Network 156 *)
PunchMasterShiftSolenoid := LeftShuttleOutput;

(* Network 157 *)
CenterPosA := CenterDiePosition[CenterShuttleIndex];

(* Network 158 *)
_e76(CLK := CHoleValve);
_e77(CLK := InCycle);
IF _e76.Q OR _e77.Q THEN ChangeCShuttle := TRUE; END_IF;

(* Network 159 *)
_e78(CLK := Step09);
CShuttleUnlatch := ChangeCShuttle AND _e78.Q;
IF ChangeCShuttle AND _e78.Q THEN ChangeCShuttle := FALSE; END_IF;

(* Network 160 *)
CenterShuttleOutput := ((CenterPosA AND CShuttleUnlatch) OR (CenterShuttleOutput AND NOT CShuttleUnlatch)) AND InCycle;

(* Network 161 *)
RightPosA := RightDiePosition[RightShuttleIndex];

(* Network 162 *)
_e79(CLK := RHoleValve);
_e80(CLK := InCycle);
IF _e79.Q OR _e80.Q THEN ChangeRShuttle := TRUE; END_IF;

(* Network 163 *)
_e81(CLK := Step09);
RShuttleUnlatch := ChangeRShuttle AND _e81.Q;
IF ChangeRShuttle AND _e81.Q THEN ChangeRShuttle := FALSE; END_IF;

(* Network 164 *)
RightShuttleOutput := ((RightPosA AND RShuttleUnlatch) OR (RightShuttleOutput AND NOT RShuttleUnlatch)) AND InCycle;

(* Network 165 *)
UncoilerRun := InCycle AND NOT InPosition1;
END_PROGRAM
```

#### Init.ld
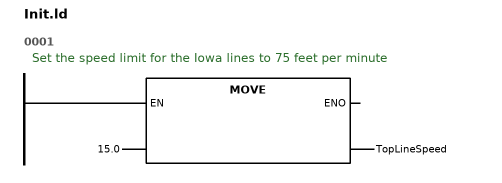
Ladder, written as Structured Text:
```iecst
PROGRAM _INIT
(* Network 1: Set the speed limit for the Iowa lines to 75 feet per minute *)
TopLineSpeed := 15.0;
END_PROGRAM
```

### Program Logical/EngelStuff (IEC) - This file handles some inputs to turn on machinery form Engel lines.

#### Variables.var
```iecst
VAR
	CLPUnlatch : BOOL;
	DuctoAutoUnlatch : BOOL;
	CEFUnlatch : BOOL;
	FullCleatUnlatch : BOOL;
	LOMUnlatch : BOOL;
	TDFUnlatch : BOOL;
	CDAUnlatch : BOOL;
END_VAR
```

#### Cyclic.ld
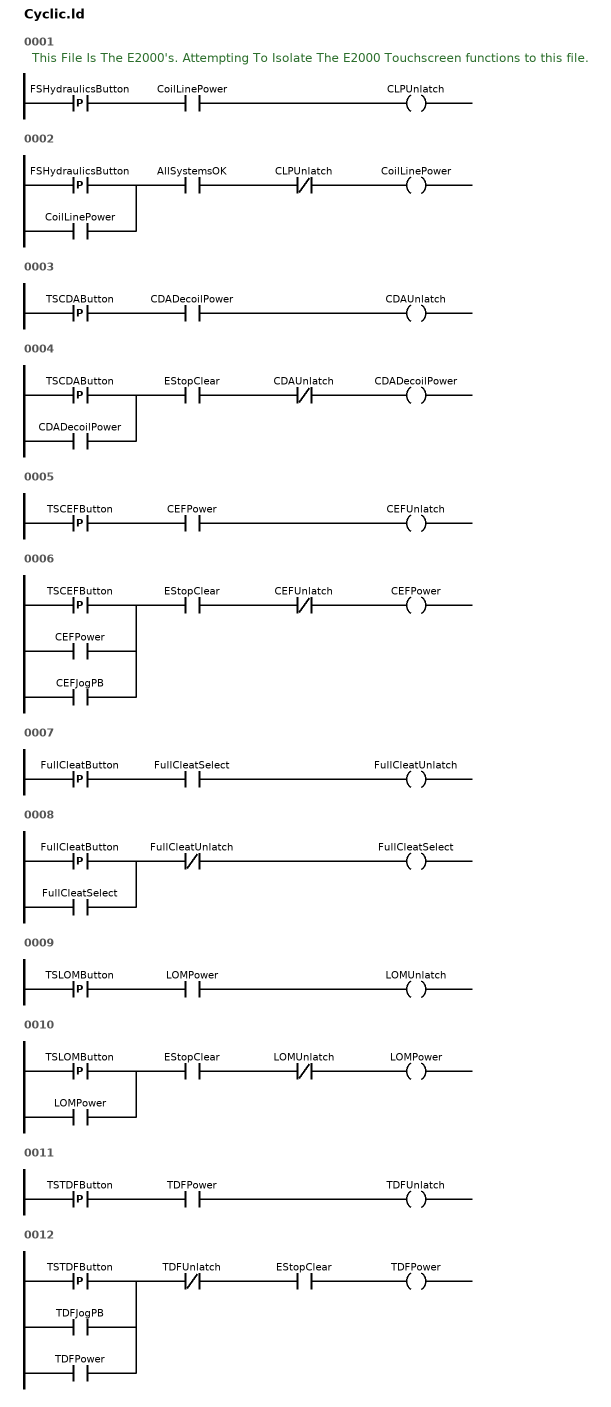
Ladder, written as Structured Text:
```iecst
PROGRAM _CYCLIC
VAR
    _e1 : R_TRIG;
    _e2 : R_TRIG;
    _e3 : R_TRIG;
    _e4 : R_TRIG;
    _e5 : R_TRIG;
    _e6 : R_TRIG;
    _e7 : R_TRIG;
    _e8 : R_TRIG;
    _e9 : R_TRIG;
    _e10 : R_TRIG;
    _e11 : R_TRIG;
    _e12 : R_TRIG;
END_VAR
(* Network 1: This File Is The E2000's. Attempting To Isolate The E2000 Touchscreen functions to this file. *)
_e1(CLK := FSHydraulicsButton);
CLPUnlatch := _e1.Q AND CoilLinePower;

(* Network 2 *)
_e2(CLK := FSHydraulicsButton);
CoilLinePower := (_e2.Q OR CoilLinePower) AND AllSystemsOK AND NOT CLPUnlatch;

(* Network 3 *)
_e3(CLK := TSCDAButton);
CDAUnlatch := _e3.Q AND CDADecoilPower;

(* Network 4 *)
_e4(CLK := TSCDAButton);
CDADecoilPower := (_e4.Q OR CDADecoilPower) AND EStopClear AND NOT CDAUnlatch;

(* Network 5 *)
_e5(CLK := TSCEFButton);
CEFUnlatch := _e5.Q AND CEFPower;

(* Network 6 *)
_e6(CLK := TSCEFButton);
CEFPower := (_e6.Q OR CEFPower OR CEFJogPB) AND EStopClear AND NOT CEFUnlatch;

(* Network 7 *)
_e7(CLK := FullCleatButton);
FullCleatUnlatch := _e7.Q AND FullCleatSelect;

(* Network 8 *)
_e8(CLK := FullCleatButton);
FullCleatSelect := (_e8.Q OR FullCleatSelect) AND NOT FullCleatUnlatch;

(* Network 9 *)
_e9(CLK := TSLOMButton);
LOMUnlatch := _e9.Q AND LOMPower;

(* Network 10 *)
_e10(CLK := TSLOMButton);
LOMPower := (_e10.Q OR LOMPower) AND EStopClear AND NOT LOMUnlatch;

(* Network 11 *)
_e11(CLK := TSTDFButton);
TDFUnlatch := _e11.Q AND TDFPower;

(* Network 12 *)
_e12(CLK := TSTDFButton);
TDFPower := (_e12.Q OR TDFJogPB OR TDFPower) AND NOT TDFUnlatch AND EStopClear;
END_PROGRAM
```

#### Init.ld
Ladder, written as Structured Text:
```iecst
PROGRAM _INIT
(* Network 1 *)
END_PROGRAM
```

### Program Logical/IMotion2 (IEC) - Engel Backgauge Wrap Brakes Motion Control Routine

#### Variables.var
```iecst
VAR
	AbsoluteDifference : DINT;
	ActualRunPercent2 : REAL;
	ActualSpeed2 : REAL;
	AMoveLength2 : DINT;
	AverageSpeed2 : REAL;
	Axis2Scaler : REAL;
	Counter2 : INT;
	DACAdd2 : REAL;
	DACBalance2 : INT;
	DecelCounter2 : INT;
	DecelDistance2 : DINT;
	DecelTime2 : REAL;
	difference : DINT;
	FirstTarget2 : BOOL;
	Hold2 : INT;
	LastPosition2 : DINT;
	MoveLength2 : DINT;
	Ratio2 : INT;
	SRM2 : REAL;
	StopWatch2 : REAL;
	TargetCount2 : INT;
	TargetDAC2 : INT;
	TopAxis2Speed : REAL := 204800;
	RealDAC2 : REAL;
	IBrakeReference : DINT;
	TopDAC2 : INT;
END_VAR
```

#### Cyclic.st
```iecst
PROGRAM _CYCLIC
	(* Electric Servo Brake Motion Control*)
	difference := IMotion2Target - (BrakeEncoder + IBrakeReference);
	AbsoluteDifference := ABS(difference);
	CASE MotionStatus2 OF
		(*Hold Position*)
		0:
			IF NOT InPosition2 THEN
				IF AbsoluteDifference <= BrakeTolerance THEN
					TargetCount2 := TargetCount2 + UpdateRate2;
					IF TargetCount2 >= SettleTime2 THEN
						InPosition2 := TRUE;
						MotionStatus2 := -1; (*Disable Drive And Put On Brake*)
					END_IF;
				END_IF;
			END_IF;

			IF (difference * 6) < MaxDAC THEN
				Ratio2 := DINT_TO_INT(difference * 6); (*Was 15 *)
			ELSE
				Ratio2 := 15000;
		    END_IF;
			IF Counter2 > 0 THEN
				Counter2 := Counter2 - UpdateRate2;
			ELSE
				Counter2 := 500;
				IF Hold2 <> Ratio2 THEN
					Hold2 := Ratio2;
				ELSE
					DACBalance2 := ActualDAC2;
				END_IF;
			END_IF;

			TargetDAC2 := Ratio2 + DACBalance2;
			ActualDAC2 := TargetDAC2;

			IF ActualDAC2 > TopDAC2 THEN
				ActualDAC2 := TopDAC2;
			END_IF;
			IF ActualDAC2 < -TopDAC2 THEN
				ActualDAC2 := -TopDAC2;
			END_IF

		(*Initialize Move*)
		1:
			Axis2Scaler := (BrakeDesired / BrakeActual);
			IMotion2Target := REAL_TO_DINT(BrakeCarriageTarget * BrakeResolution * Axis2Scaler);
			IBrakeReference := REAL_TO_DINT(BrakeReference * BrakeResolution * Axis2Scaler);
			DACAdd2 := INT_TO_REAL(MaxDAC) / AccelRampReal2;
			ActualSpeed2 := (TopAxis2Speed * DINT_TO_REAL(BackGaugeRunPercent)) / 100.0; (*Real Inches Per Second*)
			(*ActualRunPercent2 := REAL_TO_DINT(DINT_TO_REAL(BackGaugeRunPercent) / 100.0);*)
			ActualRunPercent2 := DINT_TO_REAL(BackGaugeRunPercent) / 100.0;
			TopDAC2 := REAL_TO_INT(INT_TO_REAL(MaxDAC) * ActualRunPercent2);
			IF ActualRunPercent2 = 1.0 THEN
				TopDAC2 := TopDAC2 - REAL_TO_INT(DACAdd2);
			END_IF;
			AverageSpeed2 := ActualSpeed2 / 2.0;
			DecelTime2 := (AccelRampReal2 / 1000.0) * ActualRunPercent2;
			(*DecelDistance2 := REAL_TO_DINT(((AverageSpeed2 * DecelTime2 ) * Axis2Scaler) * BrakeResolution);*)
			DecelDistance2 := REAL_TO_DINT((AverageSpeed2 * DecelTime2 ) * Axis2Scaler);
			SRM2 := MaxDACSquared / ((TopAxis2Speed * (AccelRampReal2 / 1000.0)) / 2.0);
			MoveLength2 := IMotion2Target - (BrakeEncoder + IBrakeReference);
			AMoveLength2 := ABS(MoveLength2);
			IF DecelDistance2 > (AMoveLength2 / 2) THEN
				DecelDistance2 := AMoveLength2 / 2;
				TopDAC2 := REAL_TO_INT(SQRT((DINT_TO_REAL(DecelDistance2) / Axis2Scaler) * SRM2));
				IF TopDAC2 < 3276 THEN
					TopDAC2 := 3276;
				END_IF;
			END_IF;
			InPosition2 := FALSE;
			FirstTarget2 := FALSE;
			StopWatch2 := 0.0;
			IF AMoveLength2 > REAL_TO_DINT(BrakeResolution / 16.0) THEN
				IF MoveLength2 >= 0 THEN
				  MotionStatus2 := 2;
			    ELSE
				  MotionStatus2 := 10;
				END_IF;
			ELSE
				MotionStatus2 := 12;
		    END_IF;
		(*Ramp Up To Speed*)
		2:
			IF DecelDistance2 < difference THEN
				IF ActualDAC2 < TopDAC2 THEN (*Accelerate*)
					StopWatch2 := StopWatch2 + INT_TO_REAL(UpdateRate2);
					ActualDAC2 := REAL_TO_INT(StopWatch2 * DACAdd2);
				ELSE  (*Constant Speed*)
					ActualDAC2 := TopDAC2;
				END_IF;
			ELSE (*Switch To Decel MotionState*)
				DecelCounter2 := 200;
				LastPosition2 := BrakeEncoder;
				TargetCount2 := 0;
				FirstTarget2 := FALSE	;
				MotionStatus2 := 3;
			END_IF;
		3:
			(*Stall Detection*)
			DecelCounter2 := DecelCounter2 - UpdateRate2;
			IF DecelCounter2 <= 0 THEN
				DecelCounter2 := 200;
				IF LastPosition2 = BrakeEncoder THEN
					DACBalance2 := ActualDAC2;
					Counter2 := 500;
					TopDAC2 := MaxDAC / 4;
					MotionStatus2 := 0;
				ELSE
					LastPosition2 := BrakeEncoder;
				END_IF;
			END_IF;

			RealDAC2 := REAL_TO_INT(SQRT(DINT_TO_REAL(AbsoluteDifference) * SRM2));
			IF RealDAC2 > INT_TO_REAL(MaxDAC) THEN
				RealDAC2 := INT_TO_REAL(MaxDAC);
			END_IF;
			ActualDAC2 := REAL_TO_INT(RealDAC2);

			IF FirstTarget2 THEN
				(*ActualDAC2 := ActualDAC2 / 8;*)
			END_IF;

			IF difference < 0 THEN
				ActualDAC2 := -ActualDAC2;
			END_IF;

			IF AbsoluteDifference < BrakeTolerance THEN
				FirstTarget2 := TRUE;
				TargetCount2 := TargetCount2 + UpdateRate2;
				IF TargetCount2 >= SettleTime2 THEN
					Counter2 := 500;
					InPosition2 := TRUE;
					(*MotionStatus2 := 0;*)
					MotionStatus2 := -1; (*Disable Drive And Put On Brake*)
					TopDAC2 := MaxDAC / 4;
				END_IF;
			ELSE
				TargetCount2 := 0;
			END_IF;
		4: (*Setup Forward Jog*)
			DACAdd2 := INT_TO_REAL(MaxDAC) / AccelRampReal2;
			TopDAC2 := DINT_TO_INT((INT_TO_DINT(MaxDAC) * BackGaugeJogPercent) / 100);
			TopDAC2 := TopDAC2 - REAL_TO_INT(DACAdd2);
			IBrakeReference := REAL_TO_DINT(BrakeReference * BrakeResolution * Axis2Scaler);
			StopFlag2 := FALSE;
			MotionStatus2 := 7;
		5: (*Setup Reverse Jog*)
			DACAdd2 := INT_TO_REAL(MaxDAC) / AccelRampReal2;
			TopDAC2 := DINT_TO_INT((INT_TO_DINT(MaxDAC) * BackGaugeJogPercent) / 100);
			TopDAC2 := TopDAC2 - REAL_TO_INT(DACAdd2);
			IBrakeReference := REAL_TO_DINT(BrakeReference * BrakeResolution * Axis2Scaler);
			StopFlag2 := FALSE;
			MotionStatus2 := 8;
		7: (*Forward Jog*)
			IF StopFlag2 THEN
				IF ActualDAC2 > REAL_TO_INT(DACAdd2) THEN (*Decelerate*)
					ActualDAC2 := ActualDAC2 - REAL_TO_INT(DACAdd2);
				ELSE (*Hold Position*)
					ActualDAC2 := 0;
					IMotion2Target := BrakeEncoder + IBrakeReference;
					InPosition2 := TRUE;
					MotionStatus2 := -1;
				END_IF;
			ELSE
				InPosition2 := FALSE;
				IF ActualDAC2 < TopDAC2 THEN (*Accelerate*)
					ActualDAC2 := ActualDAC2 + REAL_TO_INT(DACAdd2);
				ELSE
					ActualDAC2 := TopDAC2; (*Maintain Constant Speed*)
				END_IF;
			END_IF;
		8: (*Reverse Jog*)
			IF BackGaugeHomeLS THEN
				StopFlag2 := TRUE;
			END_IF;
			IF StopFlag2 THEN
				IF ActualDAC2 < REAL_TO_INT(-DACAdd2) THEN (*Decelerate*)
					ActualDAC2 := ActualDAC2 + REAL_TO_INT(DACAdd2);
				ELSE (*Hold Position*)
					ActualDAC2 := 0;
					IMotion2Target := BrakeEncoder + IBrakeReference;
					InPosition2 := TRUE;
					MotionStatus2 := -1;
				END_IF;
			ELSE
				InPosition1 := FALSE;
				IF ActualDAC2 > -TopDAC2 THEN (*Accelerate*)
					ActualDAC2 := ActualDAC2 - REAL_TO_INT(DACAdd2);
				ELSE
					ActualDAC2 := -TopDAC2; (*Maintain Constant Speed*)
				END_IF;
			END_IF;
		9:
			IF ActualDAC2 > REAL_TO_INT(DACAdd1) THEN (*Decelerate*)
				ActualDAC2 := ActualDAC2 - REAL_TO_INT(DACAdd2);
			ELSE (* Hold Position *)
				MetalTarget := ActlMetalEncoder;
				IncrementalRealTarget := DINT_TO_REAL(difference) / UnitsPerInch1 / MetalScaler;
				MotionStatus1 := 0;
			END_IF;
		10:
			IF DecelDistance2 < AbsoluteDifference THEN
				IF ActualDAC2 > -TopDAC2 THEN (*Accelerate*)
					StopWatch2 := StopWatch2 + INT_TO_REAL(UpdateRate2);
					ActualDAC2 := -(REAL_TO_INT(StopWatch2 * DACAdd2));
				ELSE  (*Constant Speed*)
					ActualDAC2 := -TopDAC2;
				END_IF;
			ELSE (*Switch To Decel MotionState*)
				DecelCounter2 := 200;
				LastPosition2 := BrakeEncoder;
				TargetCount2 := 0;
				FirstTarget2 := FALSE	;
				MotionStatus2 := 3;
			END_IF;
		12:
			StopWatch2 := StopWatch2 + INT_TO_REAL(UpdateRate2);
			IF StopWatch2 > 100 THEN
				InPosition2 := TRUE;
				MotionStatus2 := -1;
			END_IF;
		ELSE (*Not Moving Or Holding*)
			ActualDAC2 := 0;
			IMotion2Target := BrakeEncoder + IBrakeReference;
			InPosition2 := TRUE;
	END_CASE;

	IF ActualDAC2 > MaxDAC THEN
		ActualDAC2 := MaxDAC;
	END_IF;
	IF ActualDAC2 < -MaxDAC THEN
		ActualDAC2 := -MaxDAC;
	END_IF;

	IF MotionStatus2 >= 0 AND MotionStatus2 <> 12 THEN
		BrakeDriveEnable := TRUE;
		BackGaugeAirBrake := TRUE;
	ELSE
		BrakeDriveEnable := FALSE;
		BackGaugeAirBrake := FALSE;
	END_IF;

END_PROGRAM
```

### Program Logical/E_FWB (IEC)

#### Variables.var
```iecst
VAR
	AutoSequenceDone : BOOL;
	BAOK : BOOL;
	BCDLSDelay : BOOL;
	BDOK : BOOL;
	Bend1Required : BOOL;
	Bend2Required : BOOL;
	Bend3Required : BOOL;
	Bend4Required : BOOL;
	BendsGT0 : BOOL;
	BendsNeeded : INT;
	BHUnlatch : BOOL;
	BNIs0 : BOOL;
	BNIs1 : BOOL;
	BNIs2 : BOOL;
	BNIs3 : BOOL;
	BrakeAutoUnlatch : BOOL;
	BS : BOOL;
	BT0GT0 : BOOL;
	BT1GT0 : BOOL;
	BT2GT0 : BOOL;
	BT3GT0 : BOOL;
	ClampSettled : BOOL;
	DisableDrive : BOOL;
	FWBHome1 : BOOL;
	FWBHome2 : BOOL;
	FWBHome3 : BOOL;
	FWBHome4 : BOOL;
	FWBHome6 : BOOL;
	FWBResetTimerDone : BOOL;
	JoggingIn : BOOL;
	JoggingOut : BOOL;
	LeafSettled : BOOL;
	Look4Reset : BOOL;
	LowerBeam : BOOL;
	LowerLeaf : BOOL;
	MCPB0 : BOOL;
	MCPB1 : BOOL;
	MCPB2 : BOOL;
	MCPB3 : BOOL;
	MCPB4 : BOOL;
	MCPB5 : BOOL;
	MCPB6 : BOOL;
	MCPBTimerDone : BOOL;
	ModelIs1 : BOOL;
	OpenLatch1 : BOOL;
	PushPart : BOOL;
	PushPartUnlatch : BOOL;
	RawBrakeEncoder : REAL;
	ReadyToBend : BOOL;
	RepositionBackGauge : BOOL;
	ResOK : BOOL;
	RunSquareTimer : BOOL;
	SingleBendReset : BOOL;
	SquareArmsNotMoving : BOOL;
	SquareTmrDone : BOOL;
	StartClampTimer : BOOL;
	StartLeafTimer : BOOL;
	StartRearEject : BOOL;
	StatTimer : BOOL;
	StatTimerDone : BOOL;
	StopsDone : BOOL;
	StopsTimerDone : BOOL;
	TON_0 : TON;
	TON_1 : TON;
	TON_2 : TON;
	TON_3 : TON;
	TON_4 : TON;
	TON_5 : TON;
	TON_6 : TON;
	TON_7 : TON;
	TON_8 : TON;
	TP_0 : TP;
	TP_1 : TP;
	UnclampDelay : BOOL;
	UVDwell : BOOL;
	Wait4Move : BOOL;
	Watch4Stops : BOOL;
	xyz : BOOL;
END_VAR
```
